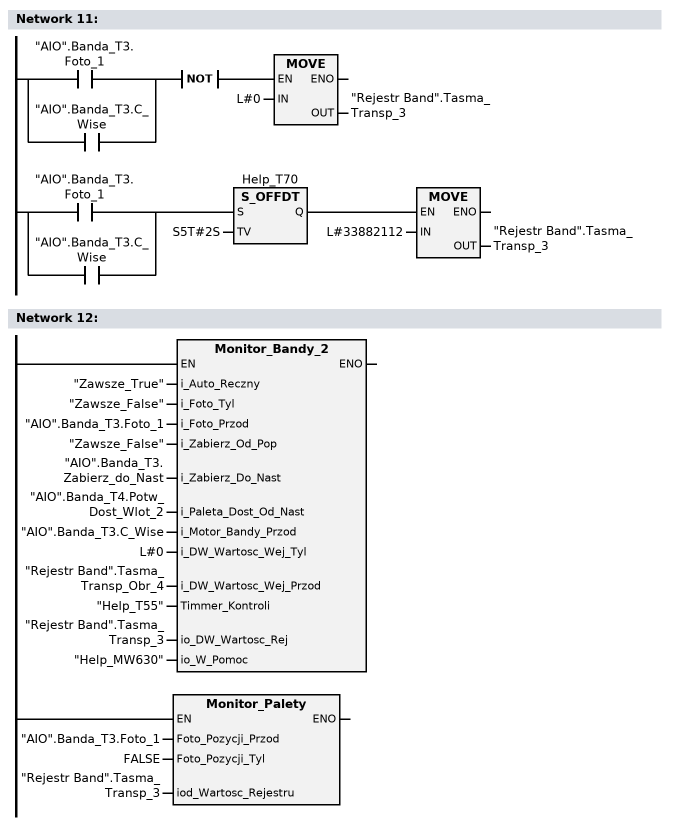
[picture p165: Monitor_Band_Lini networks 11-12]
NETWORK
TITLE =
      O     "AIO".Banda_T3.Foto_1;
      O     "AIO".Banda_T3.C_Wise;
      =     L 1.0;
      A     L 1.0;
      NOT;
      JNB   _003;
      L     L#0;
      T     "Rejestr Band".Tasma_Transp_3;
_003: NOP   0;
      A(;
      A     L 1.0;
      L     S5T#2S;
      SF    "Help_T70";
      NOP   0;
      NOP   0;
      NOP   0;
      A     "Help_T70";
      );
      JNB   _004;
      L     L#33882112;
      T     "Rejestr Band".Tasma_Transp_3;
_004: NOP   0;
NETWORK
TITLE =
//Nastepne monitoringi trzeba dopisac
//How do you do?
//Banda uznawana za wlot 2
//boczna
//Zaladauj wartosc dla wlotu jest to liczba 5 i foliowanie aktywne
//  327 680 -liczba 5
//33 882 112- liczba 5 i foliowanie   (10_0000_0101_0000_0000_0000_0000)
//**********************************************************************
      CALL  "Monitor_Bandy_2" (
           i_Auto_Reczny            := "Zawsze_True",
           i_Foto_Tyl               := "Zawsze_False",
           i_Foto_Przod             := "AIO".Banda_T3.Foto_1,
           i_Zabierz_Od_Pop         := "Zawsze_False",
           i_Zabierz_Do_Nast        := "AIO".Banda_T3.Zabierz_do_Nast,
           i_Paleta_Dost_Od_Nast    := "AIO".Banda_T4.Potw_Dost_Wlot_2,
           i_Motor_Bandy_Przod      := "AIO".Banda_T3.C_Wise,
           i_DW_Wartosc_Wej_Tyl     := L#0,
           i_DW_Wartosc_Wej_Przod   := "Rejestr Band".Tasma_Transp_Obr_4,
           Timmer_Kontroli          := "Help_T55",
           io_DW_Wartosc_Rej        := "Rejestr Band".Tasma_Transp_3,
           io_W_Pomoc               := "Help_MW630");
      CALL  "Monitor_Palety" (
           Foto_Pozycji_Przod       := "AIO".Banda_T3.Foto_1,
           Foto_Pozycji_Tyl         := FALSE,
           iod_Wartosc_Rejestru     := "Rejestr Band".Tasma_Transp_3);
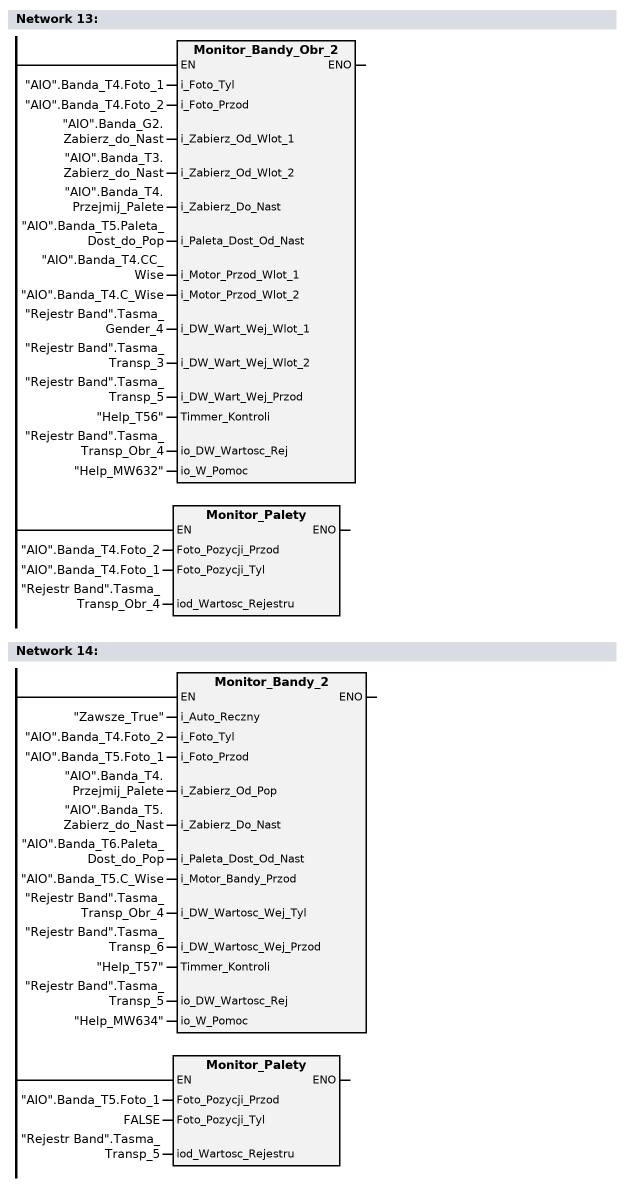
NETWORK
TITLE =
//band a obrotowa T4
//foto_2 to foto blizej foliarki
//motor prawo to motor prosto ("AIO".Banda_T4.CC_Wise)
//motor lewo to motor tyl ("AIO".Banda_T4.C_Wise)
      CALL  "Monitor_Bandy_Obr_2" (
           i_Foto_Tyl               := "AIO".Banda_T4.Foto_1,
           i_Foto_Przod             := "AIO".Banda_T4.Foto_2,
           i_Zabierz_Od_Wlot_1      := "AIO".Banda_G2.Zabierz_do_Nast,
           i_Zabierz_Od_Wlot_2      := "AIO".Banda_T3.Zabierz_do_Nast,
           i_Zabierz_Do_Nast        := "AIO".Banda_T4.Przejmij_Palete,
           i_Paleta_Dost_Od_Nast    := "AIO".Banda_T5.Paleta_Dost_do_Pop,
           i_Motor_Przod_Wlot_1     := "AIO".Banda_T4.CC_Wise,
           i_Motor_Przod_Wlot_2     := "AIO".Banda_T4.C_Wise,
           i_DW_Wart_Wej_Wlot_1     := "Rejestr Band".Tasma_Gender_4,
           i_DW_Wart_Wej_Wlot_2     := "Rejestr Band".Tasma_Transp_3,
           i_DW_Wart_Wej_Przod      := "Rejestr Band".Tasma_Transp_5,
           Timmer_Kontroli          := "Help_T56",
           io_DW_Wartosc_Rej        := "Rejestr Band".Tasma_Transp_Obr_4,
           io_W_Pomoc               := "Help_MW632");
      CALL  "Monitor_Palety" (
           Foto_Pozycji_Przod       := "AIO".Banda_T4.Foto_2,
           Foto_Pozycji_Tyl         := "AIO".Banda_T4.Foto_1,
           iod_Wartosc_Rejestru     := "Rejestr Band".Tasma_Transp_Obr_4);
NETWORK
TITLE =
//Banda T5 foto_2 na obrotnicy to ta blizej foliarki
      CALL  "Monitor_Bandy_2" (
           i_Auto_Reczny            := "Zawsze_True",
           i_Foto_Tyl               := "AIO".Banda_T4.Foto_2,
           i_Foto_Przod             := "AIO".Banda_T5.Foto_1,
           i_Zabierz_Od_Pop         := "AIO".Banda_T4.Przejmij_Palete,
           i_Zabierz_Do_Nast        := "AIO".Banda_T5.Zabierz_do_Nast,
           i_Paleta_Dost_Od_Nast    := "AIO".Banda_T6.Paleta_Dost_do_Pop,
           i_Motor_Bandy_Przod      := "AIO".Banda_T5.C_Wise,
           i_DW_Wartosc_Wej_Tyl     := "Rejestr Band".Tasma_Transp_Obr_4,
           i_DW_Wartosc_Wej_Przod   := "Rejestr Band".Tasma_Transp_6,
           Timmer_Kontroli          := "Help_T57",
           io_DW_Wartosc_Rej        := "Rejestr Band".Tasma_Transp_5,
           io_W_Pomoc               := "Help_MW634");
      CALL  "Monitor_Palety" (
           Foto_Pozycji_Przod       := "AIO".Banda_T5.Foto_1,
           Foto_Pozycji_Tyl         := FALSE,
           iod_Wartosc_Rejestru     := "Rejestr Band".Tasma_Transp_5);
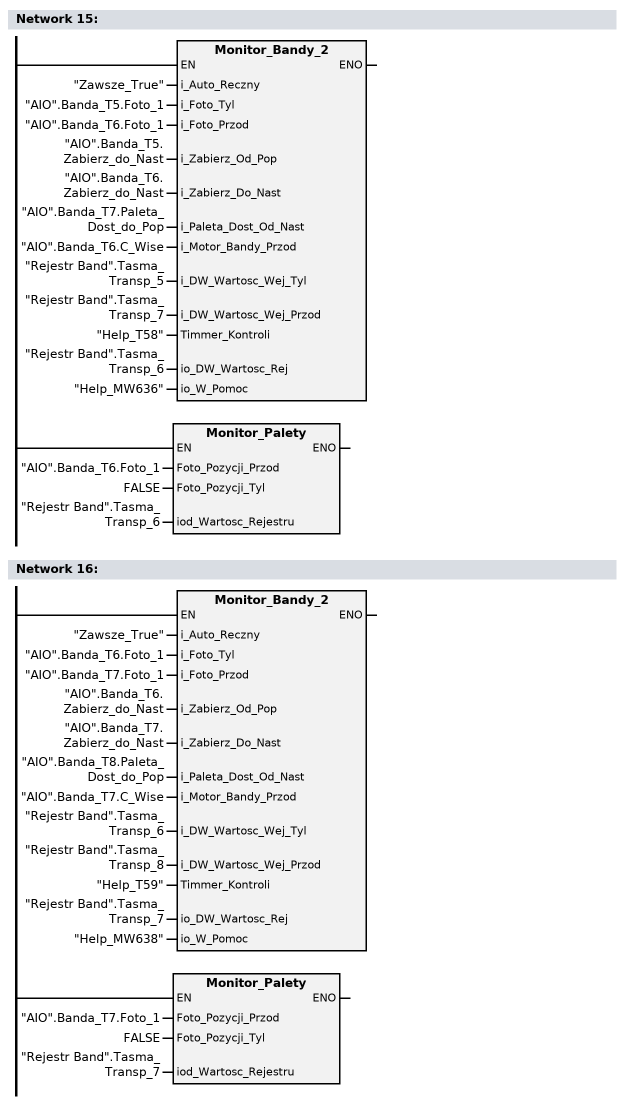
NETWORK
TITLE =
//Banda T6
      CALL  "Monitor_Bandy_2" (
           i_Auto_Reczny            := "Zawsze_True",
           i_Foto_Tyl               := "AIO".Banda_T5.Foto_1,
           i_Foto_Przod             := "AIO".Banda_T6.Foto_1,
           i_Zabierz_Od_Pop         := "AIO".Banda_T5.Zabierz_do_Nast,
           i_Zabierz_Do_Nast        := "AIO".Banda_T6.Zabierz_do_Nast,
           i_Paleta_Dost_Od_Nast    := "AIO".Banda_T7.Paleta_Dost_do_Pop,
           i_Motor_Bandy_Przod      := "AIO".Banda_T6.C_Wise,
           i_DW_Wartosc_Wej_Tyl     := "Rejestr Band".Tasma_Transp_5,
           i_DW_Wartosc_Wej_Przod   := "Rejestr Band".Tasma_Transp_7,
           Timmer_Kontroli          := "Help_T58",
           io_DW_Wartosc_Rej        := "Rejestr Band".Tasma_Transp_6,
           io_W_Pomoc               := "Help_MW636");
      CALL  "Monitor_Palety" (
           Foto_Pozycji_Przod       := "AIO".Banda_T6.Foto_1,
           Foto_Pozycji_Tyl         := FALSE,
           iod_Wartosc_Rejestru     := "Rejestr Band".Tasma_Transp_6);
NETWORK
TITLE =
//Banda T7
//
      CALL  "Monitor_Bandy_2" (
           i_Auto_Reczny            := "Zawsze_True",
           i_Foto_Tyl               := "AIO".Banda_T6.Foto_1,
           i_Foto_Przod             := "AIO".Banda_T7.Foto_1,
           i_Zabierz_Od_Pop         := "AIO".Banda_T6.Zabierz_do_Nast,
           i_Zabierz_Do_Nast        := "AIO".Banda_T7.Zabierz_do_Nast,
           i_Paleta_Dost_Od_Nast    := "AIO".Banda_T8.Paleta_Dost_do_Pop,
           i_Motor_Bandy_Przod      := "AIO".Banda_T7.C_Wise,
           i_DW_Wartosc_Wej_Tyl     := "Rejestr Band".Tasma_Transp_6,
           i_DW_Wartosc_Wej_Przod   := "Rejestr Band".Tasma_Transp_8,
           Timmer_Kontroli          := "Help_T59",
           io_DW_Wartosc_Rej        := "Rejestr Band".Tasma_Transp_7,
           io_W_Pomoc               := "Help_MW638");
      CALL  "Monitor_Palety" (
           Foto_Pozycji_Przod       := "AIO".Banda_T7.Foto_1,
           Foto_Pozycji_Tyl         := FALSE,
           iod_Wartosc_Rejestru     := "Rejestr Band".Tasma_Transp_7);
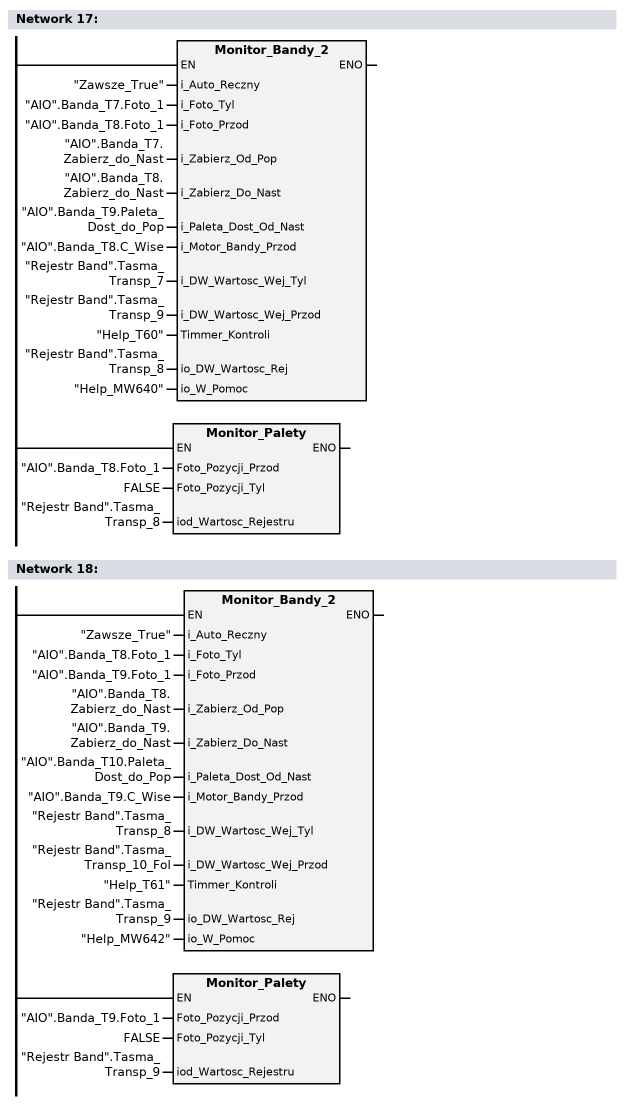
NETWORK
TITLE =
//Banda T8
//
      CALL  "Monitor_Bandy_2" (
           i_Auto_Reczny            := "Zawsze_True",
           i_Foto_Tyl               := "AIO".Banda_T7.Foto_1,
           i_Foto_Przod             := "AIO".Banda_T8.Foto_1,
           i_Zabierz_Od_Pop         := "AIO".Banda_T7.Zabierz_do_Nast,
           i_Zabierz_Do_Nast        := "AIO".Banda_T8.Zabierz_do_Nast,
           i_Paleta_Dost_Od_Nast    := "AIO".Banda_T9.Paleta_Dost_do_Pop,
           i_Motor_Bandy_Przod      := "AIO".Banda_T8.C_Wise,
           i_DW_Wartosc_Wej_Tyl     := "Rejestr Band".Tasma_Transp_7,
           i_DW_Wartosc_Wej_Przod   := "Rejestr Band".Tasma_Transp_9,
           Timmer_Kontroli          := "Help_T60",
           io_DW_Wartosc_Rej        := "Rejestr Band".Tasma_Transp_8,
           io_W_Pomoc               := "Help_MW640");
      CALL  "Monitor_Palety" (
           Foto_Pozycji_Przod       := "AIO".Banda_T8.Foto_1,
           Foto_Pozycji_Tyl         := FALSE,
           iod_Wartosc_Rejestru     := "Rejestr Band".Tasma_Transp_8);
NETWORK
TITLE =
//Banda T9
//
      CALL  "Monitor_Bandy_2" (
           i_Auto_Reczny            := "Zawsze_True",
           i_Foto_Tyl               := "AIO".Banda_T8.Foto_1,
           i_Foto_Przod             := "AIO".Banda_T9.Foto_1,
           i_Zabierz_Od_Pop         := "AIO".Banda_T8.Zabierz_do_Nast,
           i_Zabierz_Do_Nast        := "AIO".Banda_T9.Zabierz_do_Nast,
           i_Paleta_Dost_Od_Nast    := "AIO".Banda_T10.Paleta_Dost_do_Pop,
           i_Motor_Bandy_Przod      := "AIO".Banda_T9.C_Wise,
           i_DW_Wartosc_Wej_Tyl     := "Rejestr Band".Tasma_Transp_8,
           i_DW_Wartosc_Wej_Przod   := "Rejestr Band".Tasma_Transp_10_Fol,
           Timmer_Kontroli          := "Help_T61",
           io_DW_Wartosc_Rej        := "Rejestr Band".Tasma_Transp_9,
           io_W_Pomoc               := "Help_MW642");
      CALL  "Monitor_Palety" (
           Foto_Pozycji_Przod       := "AIO".Banda_T9.Foto_1,
           Foto_Pozycji_Tyl         := FALSE,
           iod_Wartosc_Rejestru     := "Rejestr Band".Tasma_Transp_9);
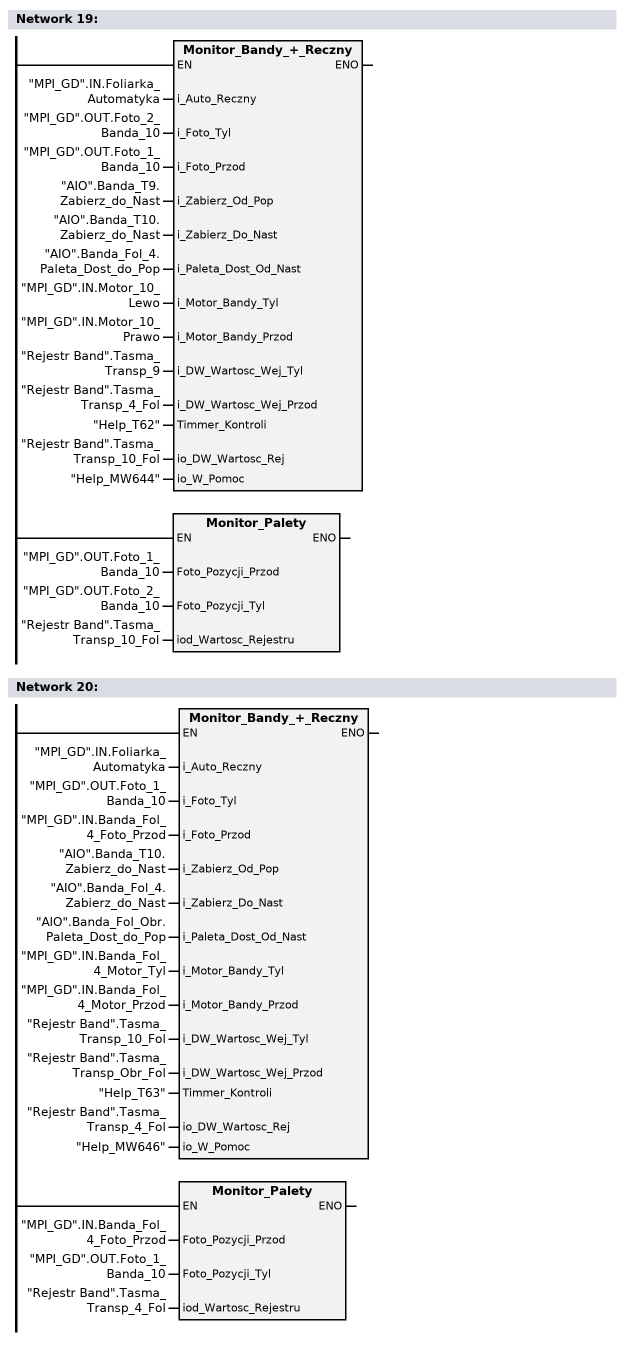
NETWORK
TITLE =
//Banda T10 - Banda 2 foliarka (ta banda jest wspolna dla lini transportowej i 
//foliarki)
//
//
//
      CALL  "Monitor_Bandy_+_Reczny" (
           i_Auto_Reczny            := "MPI_GD".IN.Foliarka_Automatyka,
           i_Foto_Tyl               := "MPI_GD".OUT.Foto_2_Banda_10,
           i_Foto_Przod             := "MPI_GD".OUT.Foto_1_Banda_10,
           i_Zabierz_Od_Pop         := "AIO".Banda_T9.Zabierz_do_Nast,
           i_Zabierz_Do_Nast        := "AIO".Banda_T10.Zabierz_do_Nast,
           i_Paleta_Dost_Od_Nast    := "AIO".Banda_Fol_4.Paleta_Dost_do_Pop,
           i_Motor_Bandy_Tyl        := "MPI_GD".IN.Motor_10_Lewo,
           i_Motor_Bandy_Przod      := "MPI_GD".IN.Motor_10_Prawo,
           i_DW_Wartosc_Wej_Tyl     := "Rejestr Band".Tasma_Transp_9,
           i_DW_Wartosc_Wej_Przod   := "Rejestr Band".Tasma_Transp_4_Fol,
           Timmer_Kontroli          := "Help_T62",
           io_DW_Wartosc_Rej        := "Rejestr Band".Tasma_Transp_10_Fol,
           io_W_Pomoc               := "Help_MW644");
      CALL  "Monitor_Palety" (
           Foto_Pozycji_Przod       := "MPI_GD".OUT.Foto_1_Banda_10,
           Foto_Pozycji_Tyl         := "MPI_GD".OUT.Foto_2_Banda_10,
           iod_Wartosc_Rejestru     := "Rejestr Band".Tasma_Transp_10_Fol);
NETWORK
TITLE =
//Banda Virtulana foliarki 4
//
      CALL  "Monitor_Bandy_+_Reczny" (
           i_Auto_Reczny            := "MPI_GD".IN.Foliarka_Automatyka,
           i_Foto_Tyl               := "MPI_GD".OUT.Foto_1_Banda_10,
           i_Foto_Przod             := "MPI_GD".IN.Banda_Fol_4_Foto_Przod,
           i_Zabierz_Od_Pop         := "AIO".Banda_T10.Zabierz_do_Nast,
           i_Zabierz_Do_Nast        := "AIO".Banda_Fol_4.Zabierz_do_Nast,
           i_Paleta_Dost_Od_Nast    := "AIO".Banda_Fol_Obr.Paleta_Dost_do_Pop,
           i_Motor_Bandy_Tyl        := "MPI_GD".IN.Banda_Fol_4_Motor_Tyl,
           i_Motor_Bandy_Przod      := "MPI_GD".IN.Banda_Fol_4_Motor_Przod,
           i_DW_Wartosc_Wej_Tyl     := "Rejestr Band".Tasma_Transp_10_Fol,
           i_DW_Wartosc_Wej_Przod   := "Rejestr Band".Tasma_Transp_Obr_Fol,
           Timmer_Kontroli          := "Help_T63",
           io_DW_Wartosc_Rej        := "Rejestr Band".Tasma_Transp_4_Fol,
           io_W_Pomoc               := "Help_MW646");
      CALL  "Monitor_Palety" (
           Foto_Pozycji_Przod       := "MPI_GD".IN.Banda_Fol_4_Foto_Przod,
           Foto_Pozycji_Tyl         := "MPI_GD".OUT.Foto_1_Banda_10,
           iod_Wartosc_Rejestru     := "Rejestr Band".Tasma_Transp_4_Fol);
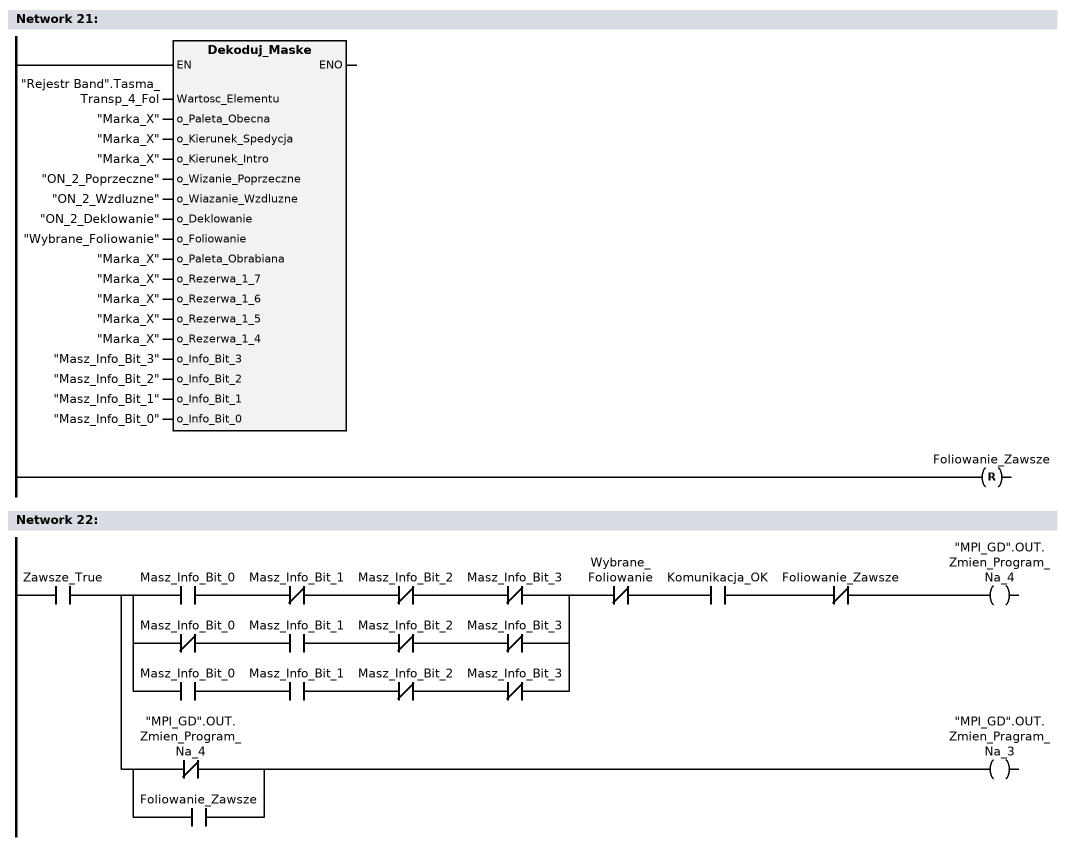
NETWORK
TITLE =
//Dekodowanie maski. Aby umozliwic bindowanie
//-Obsluga wiazan jest w FC120
//-Obsluga Dekla jest w FB3
//
      CALL  "Dekoduj_Maske" (
           Wartosc_Elementu         := "Rejestr Band".Tasma_Transp_4_Fol,
           o_Paleta_Obecna          := "Marka_X",
           o_Kierunek_Spedycja      := "Marka_X",
           o_Kierunek_Intro         := "Marka_X",
           o_Wizanie_Poprzeczne     := "ON_2_Poprzeczne",
           o_Wiazanie_Wzdluzne      := "ON_2_Wzdluzne",
           o_Deklowanie             := "ON_2_Deklowanie",
           o_Foliowanie             := "Wybrane_Foliowanie",
           o_Paleta_Obrabiana       := "Marka_X",
           o_Rezerwa_1_7            := "Marka_X",
           o_Rezerwa_1_6            := "Marka_X",
           o_Rezerwa_1_5            := "Marka_X",
           o_Rezerwa_1_4            := "Marka_X",
           o_Info_Bit_3             := "Masz_Info_Bit_3",
           o_Info_Bit_2             := "Masz_Info_Bit_2",
           o_Info_Bit_1             := "Masz_Info_Bit_1",
           o_Info_Bit_0             := "Masz_Info_Bit_0");
//Zmien program na program 4
      SET;
      R     "Foliowanie_Zawsze";
NETWORK
TITLE =
//Wybor programu foliujacego. Przewaga foliowania nad brakiem foliowania. 
//Brak foliowania wystapi jedynie gdy bedzie brak foliowania na kolbusie 1,2 oraz 
//bufforach.Po za tym paleta nie moze stracic miejsca pochodzenia
//
      A     "Zawsze_True";
      =     L 1.0;
      A     L 1.0;
      A(;
      A     "Masz_Info_Bit_0";
      AN    "Masz_Info_Bit_1";
      AN    "Masz_Info_Bit_2";
      AN    "Masz_Info_Bit_3";
      O;
      AN    "Masz_Info_Bit_0";
      A     "Masz_Info_Bit_1";
      AN    "Masz_Info_Bit_2";
      AN    "Masz_Info_Bit_3";
      O;
      A     "Masz_Info_Bit_0";
      A     "Masz_Info_Bit_1";
      AN    "Masz_Info_Bit_2";
      AN    "Masz_Info_Bit_3";
      );
      AN    "Wybrane_Foliowanie";
      A     "Komunikacja_OK";
      AN    "Foliowanie_Zawsze";
      =     "MPI_GD".OUT.Zmien_Program_Na_4;
      A     L 1.0;
      A(;
      ON    "MPI_GD".OUT.Zmien_Program_Na_4;
      O     "Foliowanie_Zawsze";
      );
      =     "MPI_GD".OUT.Zmien_Pragram_Na_3;
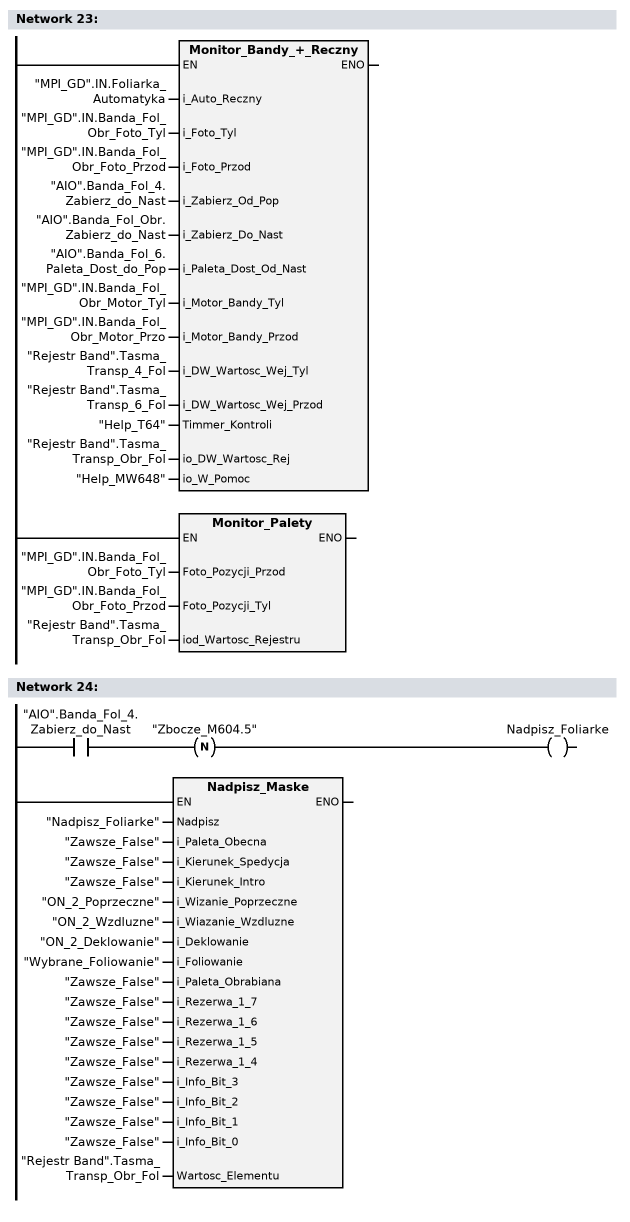
NETWORK
TITLE =
//Banda Virtulana foliarki obr
//
      CALL  "Monitor_Bandy_+_Reczny" (
           i_Auto_Reczny            := "MPI_GD".IN.Foliarka_Automatyka,
           i_Foto_Tyl               := "MPI_GD".IN.Banda_Fol_Obr_Foto_Tyl,
           i_Foto_Przod             := "MPI_GD".IN.Banda_Fol_Obr_Foto_Przod,
           i_Zabierz_Od_Pop         := "AIO".Banda_Fol_4.Zabierz_do_Nast,
           i_Zabierz_Do_Nast        := "AIO".Banda_Fol_Obr.Zabierz_do_Nast,
           i_Paleta_Dost_Od_Nast    := "AIO".Banda_Fol_6.Paleta_Dost_do_Pop,
           i_Motor_Bandy_Tyl        := "MPI_GD".IN.Banda_Fol_Obr_Motor_Tyl,
           i_Motor_Bandy_Przod      := "MPI_GD".IN.Banda_Fol_Obr_Motor_Przo,
           i_DW_Wartosc_Wej_Tyl     := "Rejestr Band".Tasma_Transp_4_Fol,
           i_DW_Wartosc_Wej_Przod   := "Rejestr Band".Tasma_Transp_6_Fol,
           Timmer_Kontroli          := "Help_T64",
           io_DW_Wartosc_Rej        := "Rejestr Band".Tasma_Transp_Obr_Fol,
           io_W_Pomoc               := "Help_MW648");
      CALL  "Monitor_Palety" (
           Foto_Pozycji_Przod       := "MPI_GD".IN.Banda_Fol_Obr_Foto_Tyl,
           Foto_Pozycji_Tyl         := "MPI_GD".IN.Banda_Fol_Obr_Foto_Przod,
           iod_Wartosc_Rejestru     := "Rejestr Band".Tasma_Transp_Obr_Fol);
NETWORK
TITLE =
//Nadpisz Maske
      A     "AIO".Banda_Fol_4.Zabierz_do_Nast;
      FN    "Zbocze_M604.5";
      =     "Nadpisz_Foliarke";
      CALL  "Nadpisz_Maske" (
           Nadpisz                  := "Nadpisz_Foliarke",
           i_Paleta_Obecna          := "Zawsze_False",
           i_Kierunek_Spedycja      := "Zawsze_False",
           i_Kierunek_Intro         := "Zawsze_False",
           i_Wizanie_Poprzeczne     := "ON_2_Poprzeczne",
           i_Wiazanie_Wzdluzne      := "ON_2_Wzdluzne",
           i_Deklowanie             := "ON_2_Deklowanie",
           i_Foliowanie             := "Wybrane_Foliowanie",
           i_Paleta_Obrabiana       := "Zawsze_False",
           i_Rezerwa_1_7            := "Zawsze_False",
           i_Rezerwa_1_6            := "Zawsze_False",
           i_Rezerwa_1_5            := "Zawsze_False",
           i_Rezerwa_1_4            := "Zawsze_False",
           i_Info_Bit_3             := "Zawsze_False",
           i_Info_Bit_2             := "Zawsze_False",
           i_Info_Bit_1             := "Zawsze_False",
           i_Info_Bit_0             := "Zawsze_False",
           Wartosc_Elementu         := "Rejestr Band".Tasma_Transp_Obr_Fol);
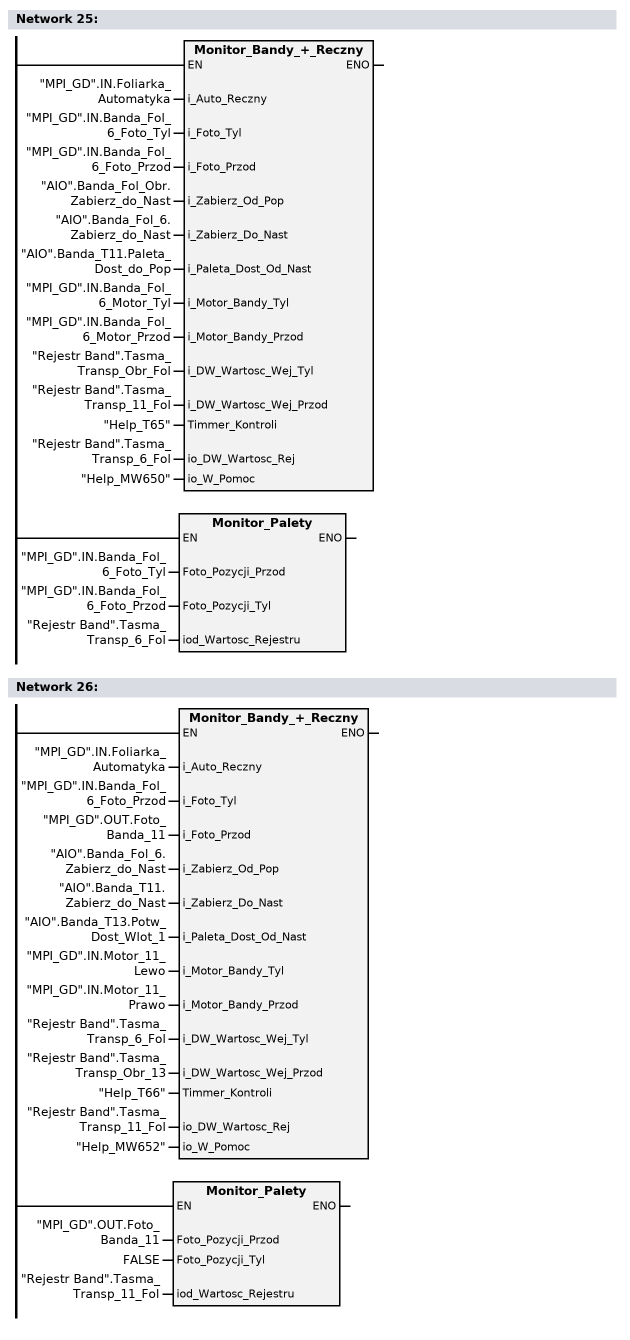
NETWORK
TITLE =
//Banda Virtulana foliarki 6
//
      CALL  "Monitor_Bandy_+_Reczny" (
           i_Auto_Reczny            := "MPI_GD".IN.Foliarka_Automatyka,
           i_Foto_Tyl               := "MPI_GD".IN.Banda_Fol_6_Foto_Tyl,
           i_Foto_Przod             := "MPI_GD".IN.Banda_Fol_6_Foto_Przod,
           i_Zabierz_Od_Pop         := "AIO".Banda_Fol_Obr.Zabierz_do_Nast,
           i_Zabierz_Do_Nast        := "AIO".Banda_Fol_6.Zabierz_do_Nast,
           i_Paleta_Dost_Od_Nast    := "AIO".Banda_T11.Paleta_Dost_do_Pop,
           i_Motor_Bandy_Tyl        := "MPI_GD".IN.Banda_Fol_6_Motor_Tyl,
           i_Motor_Bandy_Przod      := "MPI_GD".IN.Banda_Fol_6_Motor_Przod,
           i_DW_Wartosc_Wej_Tyl     := "Rejestr Band".Tasma_Transp_Obr_Fol,
           i_DW_Wartosc_Wej_Przod   := "Rejestr Band".Tasma_Transp_11_Fol,
           Timmer_Kontroli          := "Help_T65",
           io_DW_Wartosc_Rej        := "Rejestr Band".Tasma_Transp_6_Fol,
           io_W_Pomoc               := "Help_MW650");
      CALL  "Monitor_Palety" (
           Foto_Pozycji_Przod       := "MPI_GD".IN.Banda_Fol_6_Foto_Tyl,
           Foto_Pozycji_Tyl         := "MPI_GD".IN.Banda_Fol_6_Foto_Przod,
           iod_Wartosc_Rejestru     := "Rejestr Band".Tasma_Transp_6_Fol);
NETWORK
TITLE =
//Banda foliarki 11 wspolna z linia
//
      CALL  "Monitor_Bandy_+_Reczny" (
           i_Auto_Reczny            := "MPI_GD".IN.Foliarka_Automatyka,
           i_Foto_Tyl               := "MPI_GD".IN.Banda_Fol_6_Foto_Przod,
           i_Foto_Przod             := "MPI_GD".OUT.Foto_Banda_11,
           i_Zabierz_Od_Pop         := "AIO".Banda_Fol_6.Zabierz_do_Nast,
           i_Zabierz_Do_Nast        := "AIO".Banda_T11.Zabierz_do_Nast,
           i_Paleta_Dost_Od_Nast    := "AIO".Banda_T13.Potw_Dost_Wlot_1,
           i_Motor_Bandy_Tyl        := "MPI_GD".IN.Motor_11_Lewo,
           i_Motor_Bandy_Przod      := "MPI_GD".IN.Motor_11_Prawo,
           i_DW_Wartosc_Wej_Tyl     := "Rejestr Band".Tasma_Transp_6_Fol,
           i_DW_Wartosc_Wej_Przod   := "Rejestr Band".Tasma_Transp_Obr_13,
           Timmer_Kontroli          := "Help_T66",
           io_DW_Wartosc_Rej        := "Rejestr Band".Tasma_Transp_11_Fol,
           io_W_Pomoc               := "Help_MW652");
      CALL  "Monitor_Palety" (
           Foto_Pozycji_Przod       := "MPI_GD".OUT.Foto_Banda_11,
           Foto_Pozycji_Tyl         := FALSE,
           iod_Wartosc_Rejestru     := "Rejestr Band".Tasma_Transp_11_Fol);
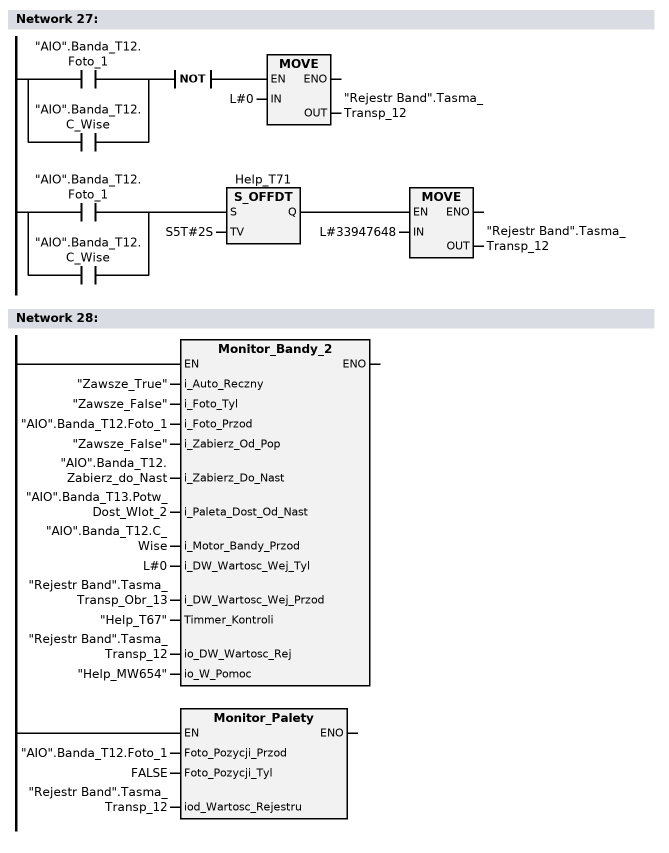
NETWORK
TITLE =
      O     "AIO".Banda_T12.Foto_1;
      O     "AIO".Banda_T12.C_Wise;
      =     L 1.0;
      A     L 1.0;
      NOT;
      JNB   _005;
      L     L#0;
      T     "Rejestr Band".Tasma_Transp_12;
_005: NOP   0;
      A(;
      A     L 1.0;
      L     S5T#2S;
      SF    "Help_T71";
      NOP   0;
      NOP   0;
      NOP   0;
      A     "Help_T71";
      );
      JNB   _006;
      L     L#33947648;
      T     "Rejestr Band".Tasma_Transp_12;
_006: NOP   0;
NETWORK
TITLE =
//Nastepne monitoringi trzeba dopisac
//Banda uznawana za wlot 3
//boczna
//Zaladauj wartosc dla wlotu jest to liczba 5 i foliowanie aktywne
//33 947 648- liczba 6 i foliowanie   (10_0000_0110_0000_0000_0000_0000)
//**********************************************************************
      CALL  "Monitor_Bandy_2" (
           i_Auto_Reczny            := "Zawsze_True",
           i_Foto_Tyl               := "Zawsze_False",
           i_Foto_Przod             := "AIO".Banda_T12.Foto_1,
           i_Zabierz_Od_Pop         := "Zawsze_False",
           i_Zabierz_Do_Nast        := "AIO".Banda_T12.Zabierz_do_Nast,
           i_Paleta_Dost_Od_Nast    := "AIO".Banda_T13.Potw_Dost_Wlot_2,
           i_Motor_Bandy_Przod      := "AIO".Banda_T12.C_Wise,
           i_DW_Wartosc_Wej_Tyl     := L#0,
           i_DW_Wartosc_Wej_Przod   := "Rejestr Band".Tasma_Transp_Obr_13,
           Timmer_Kontroli          := "Help_T67",
           io_DW_Wartosc_Rej        := "Rejestr Band".Tasma_Transp_12,
           io_W_Pomoc               := "Help_MW654");
      CALL  "Monitor_Palety" (
           Foto_Pozycji_Przod       := "AIO".Banda_T12.Foto_1,
           Foto_Pozycji_Tyl         := FALSE,
           iod_Wartosc_Rejestru     := "Rejestr Band".Tasma_Transp_12);
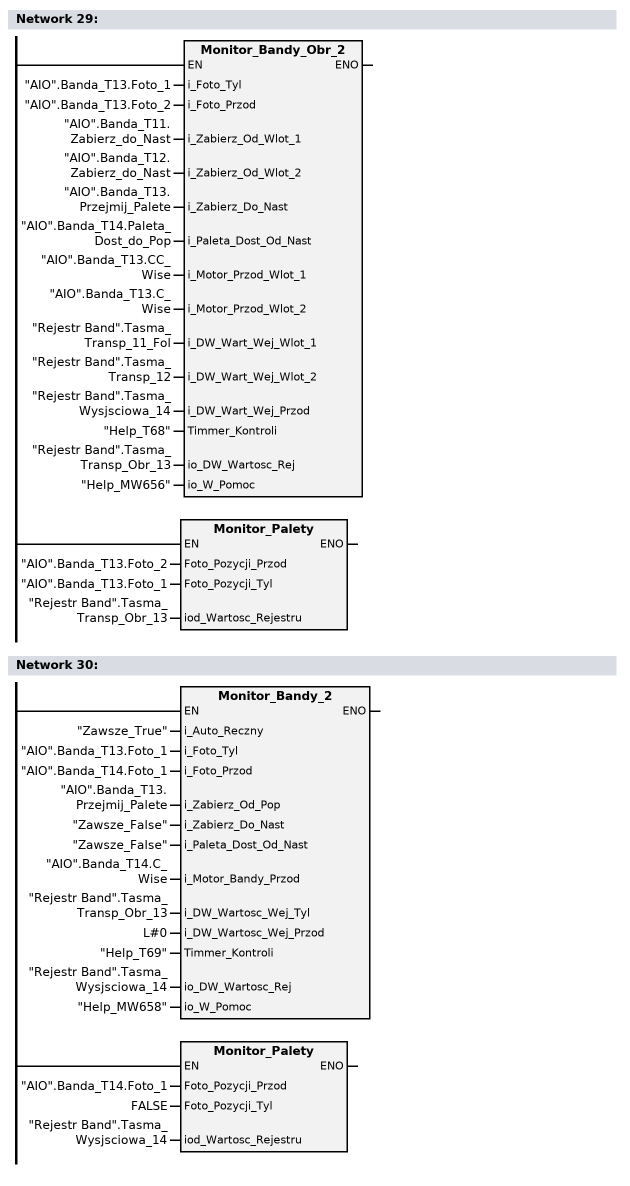
NETWORK
TITLE =
//Banda Obrotowa
//foto_2 to przod od foliarki i motor prawo
      CALL  "Monitor_Bandy_Obr_2" (
           i_Foto_Tyl               := "AIO".Banda_T13.Foto_1,
           i_Foto_Przod             := "AIO".Banda_T13.Foto_2,
           i_Zabierz_Od_Wlot_1      := "AIO".Banda_T11.Zabierz_do_Nast,
           i_Zabierz_Od_Wlot_2      := "AIO".Banda_T12.Zabierz_do_Nast,
           i_Zabierz_Do_Nast        := "AIO".Banda_T13.Przejmij_Palete,
           i_Paleta_Dost_Od_Nast    := "AIO".Banda_T14.Paleta_Dost_do_Pop,
           i_Motor_Przod_Wlot_1     := "AIO".Banda_T13.CC_Wise,
           i_Motor_Przod_Wlot_2     := "AIO".Banda_T13.C_Wise,
           i_DW_Wart_Wej_Wlot_1     := "Rejestr Band".Tasma_Transp_11_Fol,
           i_DW_Wart_Wej_Wlot_2     := "Rejestr Band".Tasma_Transp_12,
           i_DW_Wart_Wej_Przod      := "Rejestr Band".Tasma_Wysjsciowa_14,
           Timmer_Kontroli          := "Help_T68",
           io_DW_Wartosc_Rej        := "Rejestr Band".Tasma_Transp_Obr_13,
           io_W_Pomoc               := "Help_MW656");
      CALL  "Monitor_Palety" (
           Foto_Pozycji_Przod       := "AIO".Banda_T13.Foto_2,
           Foto_Pozycji_Tyl         := "AIO".Banda_T13.Foto_1,
           iod_Wartosc_Rejestru     := "Rejestr Band".Tasma_Transp_Obr_13);
NETWORK
TITLE =
//Banda Wyjsciowa ostatnia. Danke schon.
      CALL  "Monitor_Bandy_2" (
           i_Auto_Reczny            := "Zawsze_True",
           i_Foto_Tyl               := "AIO".Banda_T13.Foto_1,
           i_Foto_Przod             := "AIO".Banda_T14.Foto_1,
           i_Zabierz_Od_Pop         := "AIO".Banda_T13.Przejmij_Palete,
           i_Zabierz_Do_Nast        := "Zawsze_False",
           i_Paleta_Dost_Od_Nast    := "Zawsze_False",
           i_Motor_Bandy_Przod      := "AIO".Banda_T14.C_Wise,
           i_DW_Wartosc_Wej_Tyl     := "Rejestr Band".Tasma_Transp_Obr_13,
           i_DW_Wartosc_Wej_Przod   := L#0,
           Timmer_Kontroli          := "Help_T69",
           io_DW_Wartosc_Rej        := "Rejestr Band".Tasma_Wysjsciowa_14,
           io_W_Pomoc               := "Help_MW658");
      CALL  "Monitor_Palety" (
           Foto_Pozycji_Przod       := "AIO".Banda_T14.Foto_1,
           Foto_Pozycji_Tyl         := FALSE,
           iod_Wartosc_Rejestru     := "Rejestr Band".Tasma_Wysjsciowa_14);
END_FUNCTION

FUNCTION "Monitor_Bandy" : VOID	// FC 313
//Funkcja na monitoruje przejezdzajacy miedzy bandami produkt
VERSION : 0.1
VAR_INPUT
  i_Foto_Koniec : BOOL ;
  i_Motor_Bandy : BOOL ;
  i_Zabierz_Od_Pop : BOOL ;	//Sygnal zabierz od bandy poprzedniej
  i_Zabierz_Do_Nast : BOOL ;	//Sygnal zabierz do nastepnej
  i_DW_Wartosc_Wej : DINT ;	//Wartosc wejsciowa z poprzedniej bandy
  i_Paleta_Dost_Od_Nast : BOOL ;
END_VAR
VAR_IN_OUT
  io_DW_Wartosc_Rej : DINT ;	//Wartosc bierzaca rejestru
  io_W_Pomoc : WORD ;	//Slowo pomocnicze
END_VAR
VAR_TEMP
  Rel_Z_Pop_Aktywna : BOOL ;	//Relacja z banda poprzednia jest aktywna
  Rel_Z_Nast_Aktywna : BOOL ;	//Relacja z banda nastepna jest aktywan
  Pom_LB1 : BYTE ;
  Pom_LW2 : WORD ;
  Pom_LD4 : BOOL ;
END_VAR
BEGIN
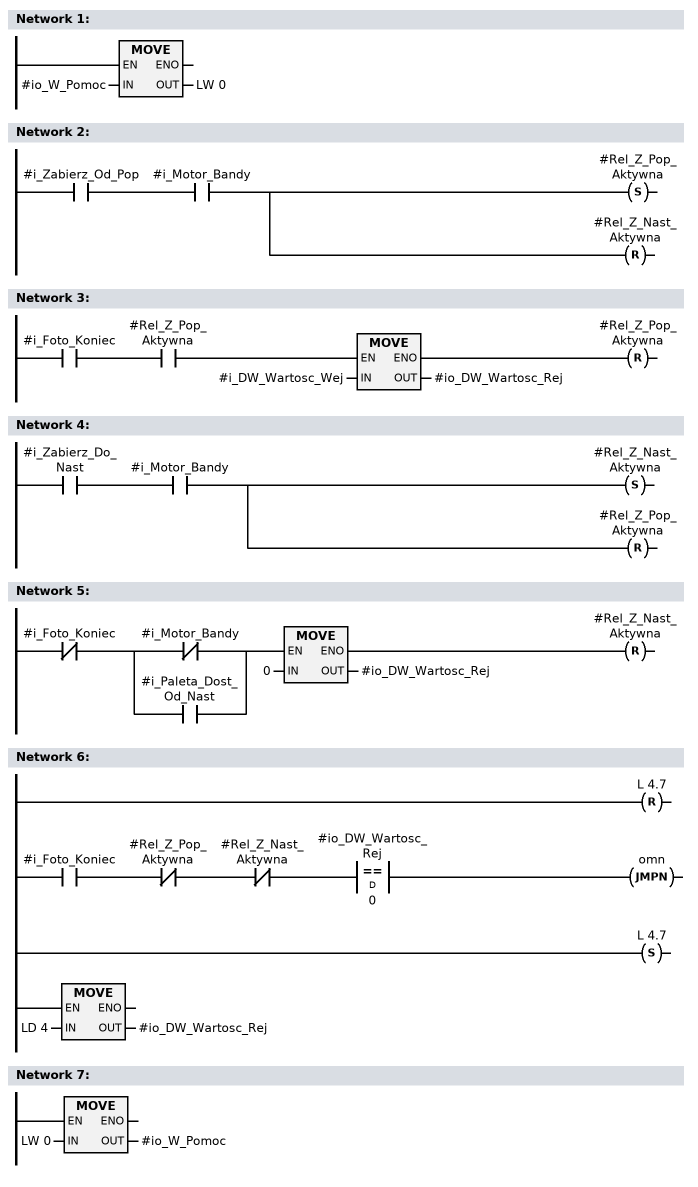
NETWORK
TITLE =
//Ten network celowo jest wolny
      L     #io_W_Pomoc;
      T     LW 0;
      NOP   0;
NETWORK
TITLE =
//Pobranie wartosci
      A     #i_Zabierz_Od_Pop;
      A     #i_Motor_Bandy;
      S     #Rel_Z_Pop_Aktywna;
      R     #Rel_Z_Nast_Aktywna;
NETWORK
TITLE =
//Dojazd do fotokomorki i przepisanie wartosci
      A     #i_Foto_Koniec;
      A     #Rel_Z_Pop_Aktywna;
      JNB   _001;
      L     #i_DW_Wartosc_Wej;
      T     #io_DW_Wartosc_Rej;
      SET;
      SAVE;
      CLR;
_001: A     BR;
      R     #Rel_Z_Pop_Aktywna;
NETWORK
TITLE =
//Relacja z nastepna banda
      A     #i_Zabierz_Do_Nast;
      A     #i_Motor_Bandy;
      S     #Rel_Z_Nast_Aktywna;
      R     #Rel_Z_Pop_Aktywna;
NETWORK
TITLE =
//Opuszczeni palety z bandy relacja przod
      AN    #i_Foto_Koniec;
      A(;
      ON    #i_Motor_Bandy;
      O     #i_Paleta_Dost_Od_Nast;
      );
      JNB   _002;
      L     0;
      T     #io_DW_Wartosc_Rej;
      SET;
      SAVE;
      CLR;
_002: A     BR;
      R     #Rel_Z_Nast_Aktywna;
NETWORK
TITLE =
//Nalozenie maski gdy jest paleta a wartosc rejsetru wskazuje na 0
//kasowanie bitu pomocniczego
      SET;
      R     L 4.7;
// Aby znalezc palete widmo
      A     #i_Foto_Koniec;
      AN    #Rel_Z_Pop_Aktywna;
      AN    #Rel_Z_Nast_Aktywna;
      A(;
      L     #io_DW_Wartosc_Rej;
      L     0;
      ==D;
      );
      JCN   omn;
      SET;
      S     L 4.7;	//najstarszy bit (info o palecie)
      L     LD 4;
      T     #io_DW_Wartosc_Rej;
omn:  NOP   0;
NETWORK
TITLE =
//Przypisanie wartosci z pamieci podrecznej
//
      L     LW 0;
      T     #io_W_Pomoc;
      NOP   0;
END_FUNCTION

FUNCTION "Monitor_Bandy_Obr" : VOID	// FC 314
//Funkcja na monitoruje przejezdzajacy miedzy bandami produkt
VERSION : 0.1
VAR_INPUT
  i_Foto_Koniec_Wlot_1 : BOOL ;
  i_Foto_Koniec_Wlot_2 : BOOL ;
  i_Foto_Koniec_Wylot : BOOL ;
  i_Motor_Bandy : BOOL ;
  i_Zabierz_Od_Wlot_1 : BOOL ;	//Sygnal zabierz od bandy poprzedniej
  i_Zabierz_Od_Wlot_2 : BOOL ;	//Sygnal zabierz od bandy poprzedniej
  i_Zabierz_Do_Nast : BOOL ;	//Sygnal zabierz do nastepnej
  i_DW_Wart_Wej_Wlot_1 : DINT ;	//Wartosc wejsciowa z wlotu 1
  i_DW_Wart_Wej_Wlot_2 : DINT ;	//Wartosc wejsciowa z wlotu 2
  i_Paleta_Dost_Od_Nast : BOOL ;
END_VAR
VAR_IN_OUT
  io_DW_Wartosc_Rej : DINT ;	//Wartosc bierzaca rejestru
  io_W_Pomoc : WORD ;	//Slowo pomocnicze
END_VAR
VAR_TEMP
  Rel_Aktyw_z_Wlot_1 : BOOL ;	//Relacja z banda poprzednia jest aktywna
  Rel_Aktyw_z_Wlot_2 : BOOL ;	//Relacja z banda poprzednia jest aktywna
  Rel_Z_Nast_Aktywna : BOOL ;	//Relacja z banda nastepna jest aktywan
  Pom_LB1 : BYTE ;
  Pom_LW2 : WORD ;
  Pom_LD4 : DINT ;
END_VAR
BEGIN
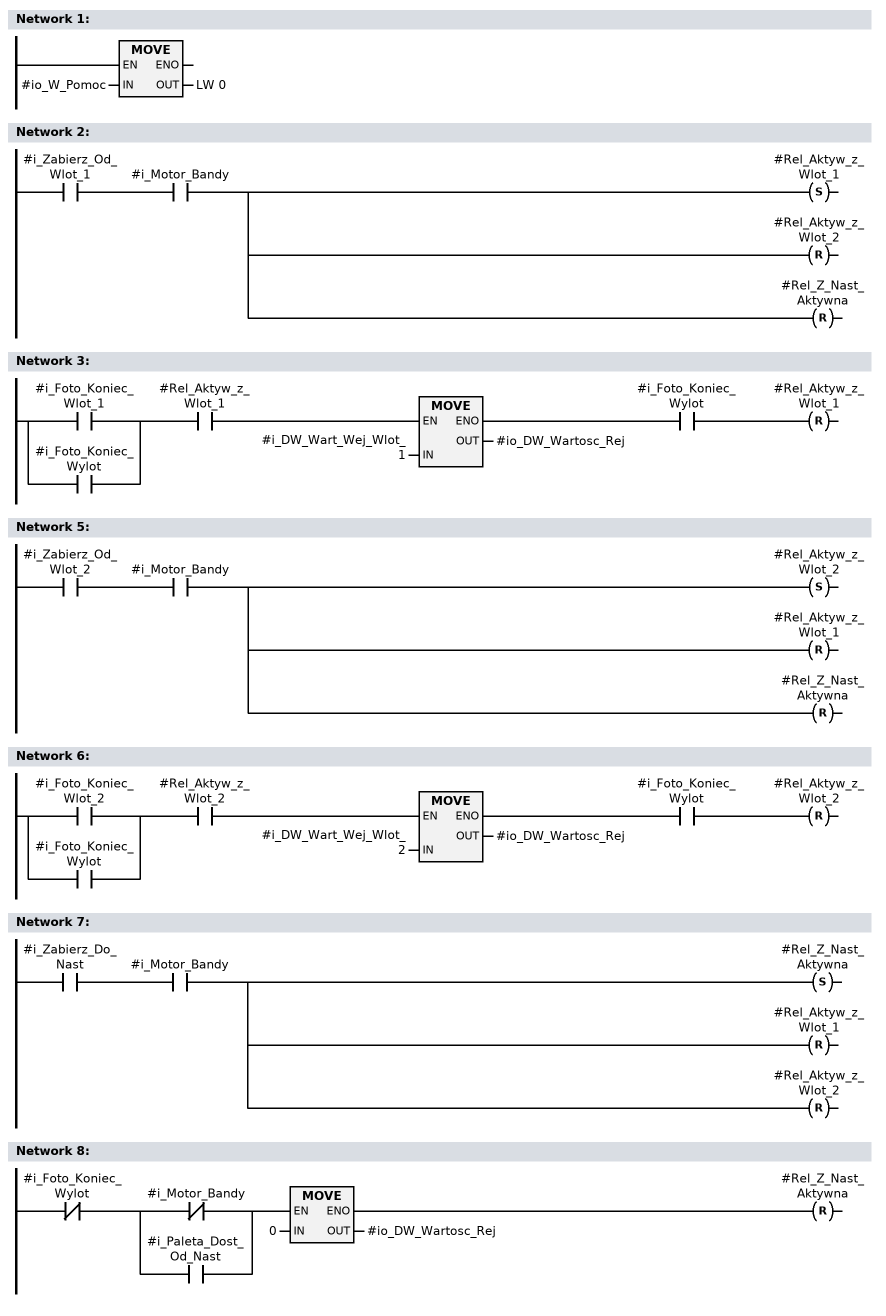
NETWORK
TITLE =
//Ten network celowo jest wolny
      L     #io_W_Pomoc;
      T     LW 0;
      NOP   0;
NETWORK
TITLE =
//Sprawdzenie Relacji z wolotem nr 1
      A     #i_Zabierz_Od_Wlot_1;
      A     #i_Motor_Bandy;
      S     #Rel_Aktyw_z_Wlot_1;
      R     #Rel_Aktyw_z_Wlot_2;
      R     #Rel_Z_Nast_Aktywna;
NETWORK
TITLE =
//Dojazd do fotokomorki i przepisanie wartosci
      A(;
      A(;
      O     #i_Foto_Koniec_Wlot_1;
      O     #i_Foto_Koniec_Wylot;
      );
      A     #Rel_Aktyw_z_Wlot_1;
      JNB   _001;
      L     #i_DW_Wart_Wej_Wlot_1;
      T     #io_DW_Wartosc_Rej;
      SET;
      SAVE;
      CLR;
_001: A     BR;
      );
      A     #i_Foto_Koniec_Wylot;
      R     #Rel_Aktyw_z_Wlot_1;
NETWORK
TITLE =
//Relacja z wlotem nr 2
NETWORK
TITLE =
//Sprawdzenie Relacji z wolotem nr 2
      A     #i_Zabierz_Od_Wlot_2;
      A     #i_Motor_Bandy;
      S     #Rel_Aktyw_z_Wlot_2;
      R     #Rel_Aktyw_z_Wlot_1;
      R     #Rel_Z_Nast_Aktywna;
NETWORK
TITLE =
//Dojazd do fotokomorki i przepisanie wartosci
      A(;
      A(;
      O     #i_Foto_Koniec_Wlot_2;
      O     #i_Foto_Koniec_Wylot;
      );
      A     #Rel_Aktyw_z_Wlot_2;
      JNB   _002;
      L     #i_DW_Wart_Wej_Wlot_2;
      T     #io_DW_Wartosc_Rej;
      SET;
      SAVE;
      CLR;
_002: A     BR;
      );
      A     #i_Foto_Koniec_Wylot;
      R     #Rel_Aktyw_z_Wlot_2;
NETWORK
TITLE =
//Relacja z nastepna banda
      A     #i_Zabierz_Do_Nast;
      A     #i_Motor_Bandy;
      S     #Rel_Z_Nast_Aktywna;
      R     #Rel_Aktyw_z_Wlot_1;
      R     #Rel_Aktyw_z_Wlot_2;
NETWORK
TITLE =
//Opuszczeni palety z bandy relacja przod
      AN    #i_Foto_Koniec_Wylot;
      A(;
      ON    #i_Motor_Bandy;
      O     #i_Paleta_Dost_Od_Nast;
      );
      JNB   _003;
      L     0;
      T     #io_DW_Wartosc_Rej;
      SET;
      SAVE;
      CLR;
_003: A     BR;
      R     #Rel_Z_Nast_Aktywna;
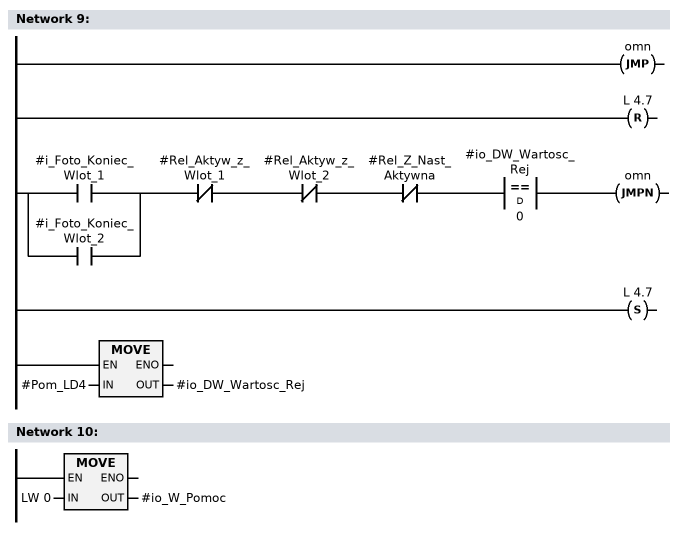
NETWORK
TITLE =
//Nalozenie maski gdy jest paleta a wartosc rejsetru wskazuje na 0
//kasowanie bitu pomocniczego
      JU    omn;
      SET;
      R     L 4.7;
// Aby znalezc palete widmo
      A(;
      O     #i_Foto_Koniec_Wlot_1;
      O     #i_Foto_Koniec_Wlot_2;
      );
      AN    #Rel_Aktyw_z_Wlot_1;
      AN    #Rel_Aktyw_z_Wlot_2;
      AN    #Rel_Z_Nast_Aktywna;
      A(;
      L     #io_DW_Wartosc_Rej;
      L     0;
      ==D;
      );
      JCN   omn;
      SET;
      S     L 4.7;	//najstarszy bit (info o palecie)
      L     #Pom_LD4;
      T     #io_DW_Wartosc_Rej;
omn:  NOP   0;
NETWORK
TITLE =
//Przypisanie wartosci z pamieci podrecznej
//
      L     LW 0;
      T     #io_W_Pomoc;
      NOP   0;
END_FUNCTION

FUNCTION "Monitor_Bandy_+_Reczny" : VOID	// FC 315
//Funkcja na monitoruje przejezdzajacy miedzy bandami produkt
//Jezeli cos nie wyjdzie paleta widmo bierze wszystko na siebie
//
//
//0.7 - paleta obecna (nieuzywane)
//0.6 - kierunek spedycja (uzywane)
//0.5 - kierunek intro (uzywane)
//0.4 - wiazanie poprzeczne (uzywane)
//0.3 - wiazanie wzdluzne   (uzywane)
//0.2 - deklowanie (uzywane)
//0.1 - foliowanie (uzywane)
//0.0 - paleta obrabiana
//1.7 - rezerwa (nieuzywane)
//1.6 - rezerwa (nieuzywane)
//1.5 - rezerwa (nieuzywane)
//1.3 - rezerwa (nieuzywane)
//1.3 - info bit 3
//1.2 - info bit 2
//1.1 - info bit 1 
//1.0 - info bit 0
//
VERSION : 0.1
VAR_INPUT
  i_Auto_Reczny : BOOL ;	//1-Auto; 0-Reczny
  i_Foto_Tyl : BOOL ;
  i_Foto_Przod : BOOL ;
  i_Zabierz_Od_Pop : BOOL ;	//Sygnal zabierz od bandy poprzedniej
  i_Zabierz_Do_Nast : BOOL ;	//Sygnal zabierz do nastepnej
  i_Paleta_Dost_Od_Nast : BOOL ;
  i_Motor_Bandy_Tyl : BOOL ;
  i_Motor_Bandy_Przod : BOOL ;
  i_DW_Wartosc_Wej_Tyl : DINT ;	//Wartosc wejsciowa z poprzedniej bandy
  i_DW_Wartosc_Wej_Przod : DINT ;	//Wartosc wejsciowa z poprzedniej bandy
  Timmer_Kontroli : TIMER ;
END_VAR
VAR_IN_OUT
  io_DW_Wartosc_Rej : DINT ;	//Wartosc bierzaca rejestru
  io_W_Pomoc : WORD ;	//Slowo pomocnicze
END_VAR
VAR_TEMP
  Rel_Z_Pop_Aktywna : BOOL ;	//Relacja z banda poprzednia jest aktywna
  Rel_Z_Nast_Aktywna : BOOL ;	//Relacja z banda nastepna jest aktywan
  Help_Zbocze_1 : BOOL ;
  Help_Zbocze_2 : BOOL ;
  Help_Zbocze_3 : BOOL ;
  Help_Zbocze_4 : BOOL ;
  Help_Zbocze_5 : BOOL ;
  Pom_LB1 : BYTE ;
  Pom_LW2 : WORD ;
  Pom_LD4 : DINT ;
  Pom_LD8 : DINT ;
END_VAR
BEGIN
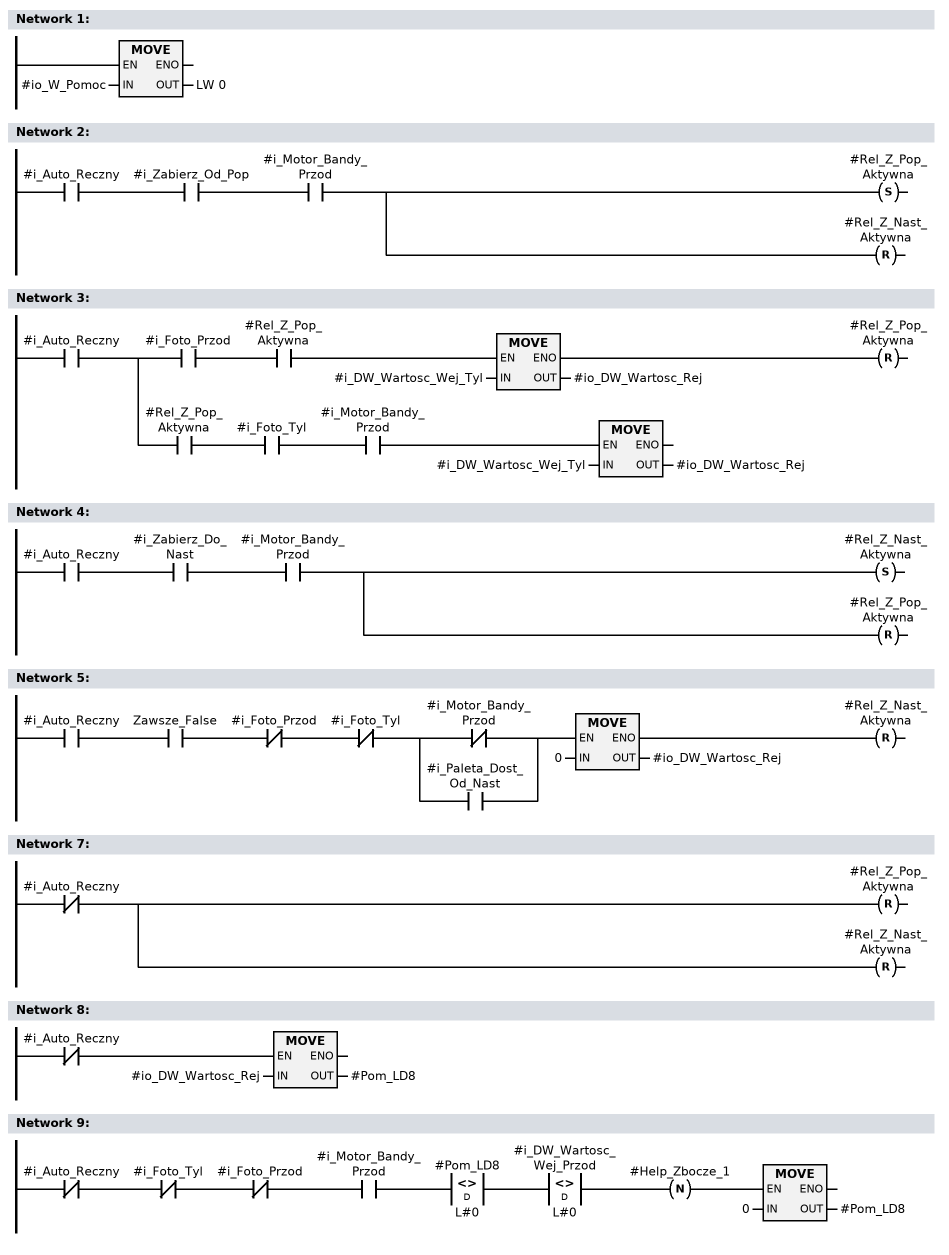
NETWORK
TITLE =
//Ten network celowo jest wolny
      L     #io_W_Pomoc;
      T     LW 0;
      NOP   0;
NETWORK
TITLE =
//Tryb Auto
//Pobranie wartosci
//
      A     #i_Auto_Reczny;
      A     #i_Zabierz_Od_Pop;
      A     #i_Motor_Bandy_Przod;
      S     #Rel_Z_Pop_Aktywna;
      R     #Rel_Z_Nast_Aktywna;
NETWORK
TITLE =
//Dojazd do fotokomorki i przepisanie wartosci.Informacja moze byc tez szybciej 
//przekazana (Gender potrzebuje szybciej)
      A     #i_Auto_Reczny;
      =     L 12.0;
      A     L 12.0;
      A     #i_Foto_Przod;
      A     #Rel_Z_Pop_Aktywna;
      JNB   _001;
      L     #i_DW_Wartosc_Wej_Tyl;
      T     #io_DW_Wartosc_Rej;
      SET;
      SAVE;
      CLR;
_001: A     BR;
      R     #Rel_Z_Pop_Aktywna;
      A     L 12.0;
      A     #Rel_Z_Pop_Aktywna;
      A     #i_Foto_Tyl;
      A     #i_Motor_Bandy_Przod;
      JNB   _002;
      L     #i_DW_Wartosc_Wej_Tyl;
      T     #io_DW_Wartosc_Rej;
_002: NOP   0;
NETWORK
TITLE =
//Relacja z nastepna banda
      A     #i_Auto_Reczny;
      A     #i_Zabierz_Do_Nast;
      A     #i_Motor_Bandy_Przod;
      S     #Rel_Z_Nast_Aktywna;
      R     #Rel_Z_Pop_Aktywna;
NETWORK
TITLE =
//Opuszczeni palety z bandy relacja przod
      A     #i_Auto_Reczny;
      A     "Zawsze_False";
      AN    #i_Foto_Przod;
      AN    #i_Foto_Tyl;
      A(;
      ON    #i_Motor_Bandy_Przod;
      O     #i_Paleta_Dost_Od_Nast;
      );
      JNB   _003;
      L     0;
      T     #io_DW_Wartosc_Rej;
      SET;
      SAVE;
      CLR;
_003: A     BR;
      R     #Rel_Z_Nast_Aktywna;
NETWORK
TITLE =
//Tryb Reczny
//Warunkiem prawidlowego dzialania trybu reczenego jest pokrycie zawsze co 
//najmniej jednej fotokomorki gdy jest produkt
//
//
NETWORK
TITLE =
//Zresetowanie relacji z automatyki
//
      AN    #i_Auto_Reczny;
      R     #Rel_Z_Pop_Aktywna;
      R     #Rel_Z_Nast_Aktywna;
NETWORK
TITLE =
//Trzeba sobie jakos radzic
      AN    #i_Auto_Reczny;
      JNB   _004;
      L     #io_DW_Wartosc_Rej;
      T     #Pom_LD8;
_004: NOP   0;
NETWORK
TITLE =
//Jazda do przodu na recznym.Bierzaca--->Nastepna
      AN    #i_Auto_Reczny;
      AN    #i_Foto_Tyl;
      AN    #i_Foto_Przod;
      A     #i_Motor_Bandy_Przod;
      A(;
      L     #Pom_LD8;
      L     L#0;
      <>D;
      );
      A(;
      L     #i_DW_Wartosc_Wej_Przod;
      L     L#0;
      <>D;
      );
      FN    #Help_Zbocze_1;
      JNB   _005;
      L     0;
      T     #Pom_LD8;
_005: NOP   0;
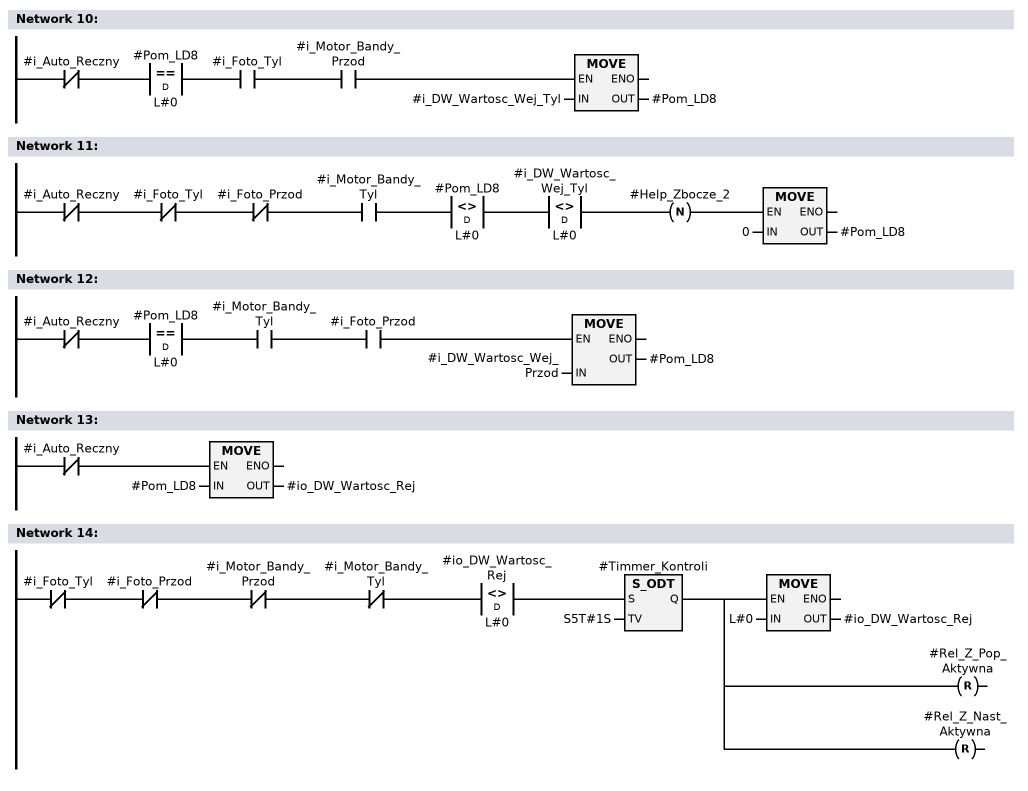
NETWORK
TITLE =
//Poprzednia wjezdza na bierzaca w trybie recznym. Poprzednia--->Bierzaca
      AN    #i_Auto_Reczny;
      A(;
      L     #Pom_LD8;
      L     L#0;
      ==D;
      );
      A     #i_Foto_Tyl;
      A     #i_Motor_Bandy_Przod;
      JNB   _006;
      L     #i_DW_Wartosc_Wej_Tyl;
      T     #Pom_LD8;
_006: NOP   0;
NETWORK
TITLE =
//Bierzaca wjezdza na bande porzedzajaca. Bierzaca--->Poprzednia
      AN    #i_Auto_Reczny;
      AN    #i_Foto_Tyl;
      AN    #i_Foto_Przod;
      A     #i_Motor_Bandy_Tyl;
      A(;
      L     #Pom_LD8;
      L     L#0;
      <>D;
      );
      A(;
      L     #i_DW_Wartosc_Wej_Tyl;
      L     L#0;
      <>D;
      );
      FN    #Help_Zbocze_2;
      JNB   _007;
      L     0;
      T     #Pom_LD8;
_007: NOP   0;
NETWORK
TITLE =
//Z Nastepnej wjezdza na bierzaca. Nastepna--->Bierzaca
      AN    #i_Auto_Reczny;
      A(;
      L     #Pom_LD8;
      L     L#0;
      ==D;
      );
      A     #i_Motor_Bandy_Tyl;
      A     #i_Foto_Przod;
      JNB   _008;
      L     #i_DW_Wartosc_Wej_Przod;
      T     #Pom_LD8;
_008: NOP   0;
NETWORK
TITLE =
//Przepisanie powrotne
      AN    #i_Auto_Reczny;
      JNB   _009;
      L     #Pom_LD8;
      T     #io_DW_Wartosc_Rej;
_009: NOP   0;
NETWORK
TITLE =
//Sprawdznie wszystkiego
//
      AN    #i_Foto_Tyl;
      AN    #i_Foto_Przod;
      AN    #i_Motor_Bandy_Przod;
      AN    #i_Motor_Bandy_Tyl;
      A(;
      L     #io_DW_Wartosc_Rej;
      L     L#0;
      <>D;
      );
      L     S5T#1S;
      SD    #Timmer_Kontroli;
      NOP   0;
      NOP   0;
      NOP   0;
      A     #Timmer_Kontroli;
      =     L 12.0;
      A     L 12.0;
      JNB   _00a;
      L     L#0;
      T     #io_DW_Wartosc_Rej;
_00a: NOP   0;
      A     L 12.0;
      BLD   102;
      R     #Rel_Z_Pop_Aktywna;
      A     L 12.0;
      BLD   102;
      R     #Rel_Z_Nast_Aktywna;
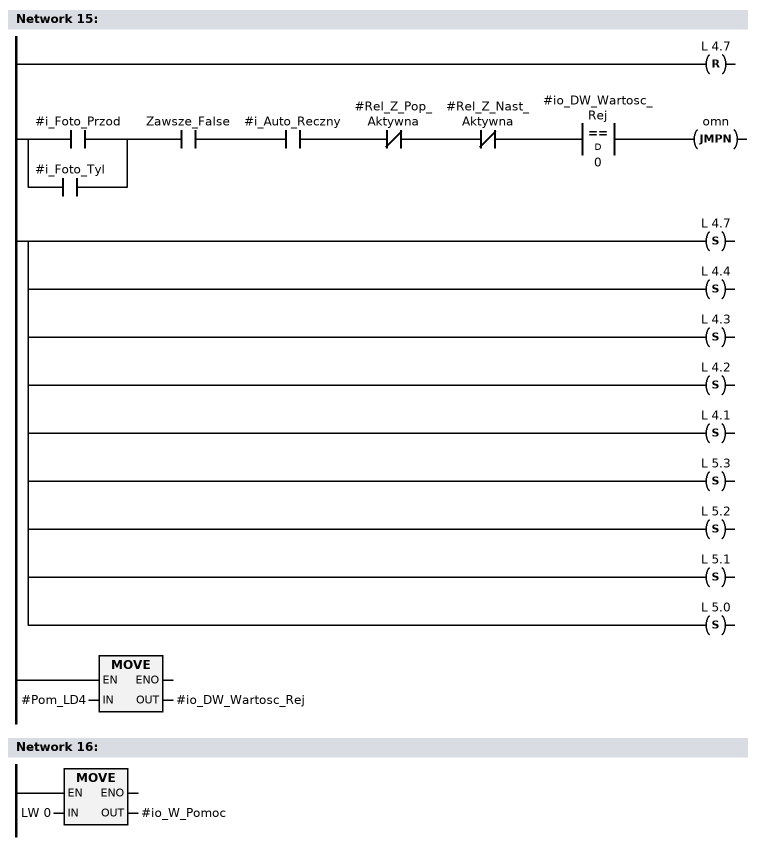
NETWORK
TITLE =
//0.7 - paleta obecna (nieuzywane)
//0.6 - kierunek spedycja (uzywane)
//0.5 - kierunek intro (uzywane)
//0.4 - wiazanie poprzeczne (uzywane)
//0.3 - wiazanie wzdluzne   (uzywane)
//0.2 - deklowanie (uzywane)
//0.1 - foliowanie (uzywane)
//0.0 - paleta obrabiana
//1.7 - rezerwa (nieuzywane)
//1.6 - rezerwa (nieuzywane)
//1.5 - rezerwa (nieuzywane)
//1.3 - rezerwa (nieuzywane)
//1.3 - info bit 3
//1.2 - info bit 2
//1.1 - info bit 1 
//1.0 - info bit 0
//
//kasowanie bitu pomocniczego
      SET;
      R     L 4.7;
// Aby znalezc palete widmo
      O     #i_Foto_Przod;
      O     #i_Foto_Tyl;
      A     "Zawsze_False";
      A     #i_Auto_Reczny;
      AN    #Rel_Z_Pop_Aktywna;
      AN    #Rel_Z_Nast_Aktywna;
      A(;
      L     #io_DW_Wartosc_Rej;
      L     0;
      ==D;
      );
      JCN   omn;
      SET;
      S     L 4.7;	//najstarszy bit (info o palecie)
      S     L 4.4;	//pop
      S     L 4.3;	//wzd
      S     L 4.2;	//dek
      S     L 4.1;	//fol
//--Daj znaczniki ze to paleta widmo
      S     L 5.3;
      S     L 5.2;
      S     L 5.1;
      S     L 5.0;
      L     #Pom_LD4;
      T     #io_DW_Wartosc_Rej;
omn:  NOP   0;
NETWORK
TITLE =
//Przypisanie wartosci z pamieci podrecznej
//
      L     LW 0;
      T     #io_W_Pomoc;
      NOP   0;
END_FUNCTION

FUNCTION "Monitor_Palety" : VOID	// FC 316
VERSION : 0.1
VAR_INPUT
  Foto_Pozycji_Przod : BOOL ;
  Foto_Pozycji_Tyl : BOOL ;	//Opcjonalna fotokomorka
END_VAR
VAR_IN_OUT
  iod_Wartosc_Rejestru : DINT ;
END_VAR
VAR_TEMP
  Wartosc_Pomocnicz_0 : DINT ;
  Wartosc_Pomocnicz_1 : DINT ;
END_VAR
BEGIN
NETWORK
TITLE =
      L     #iod_Wartosc_Rejestru;
      T     #Wartosc_Pomocnicz_0;
      O     #Foto_Pozycji_Przod;
      O     #Foto_Pozycji_Tyl;
      JCN   et_1;
      SET;
      S     L 0.7;
et_1: NOP   0;
      AN    #Foto_Pozycji_Przod;
      AN    #Foto_Pozycji_Tyl;
      JCN   et_2;
      SET;
      R     L 0.7;
et_2: NOP   0;
      L     #Wartosc_Pomocnicz_0;
      T     #iod_Wartosc_Rejestru;
END_FUNCTION

FUNCTION "Monitor_Bandy_2" : VOID	// FC 317
//Funkcja na monitoruje przejezdzajacy miedzy bandami produkt
//Jezeli cos nie wyjdzie paleta widmo bierze wszystko na siebie
//
//
//0.7 - paleta obecna (nieuzywane)
//0.6 - kierunek spedycja (uzywane)
//0.5 - kierunek intro (uzywane)
//0.4 - wiazanie poprzeczne (uzywane)
//0.3 - wiazanie wzdluzne   (uzywane)
//0.2 - deklowanie (uzywane)
//0.1 - foliowanie (uzywane)
//0.0 - paleta obrabiana
//1.7 - rezerwa (nieuzywane)
//1.6 - rezerwa (nieuzywane)
//1.5 - rezerwa (nieuzywane)
//1.3 - rezerwa (nieuzywane)
//1.3 - info bit 3
//1.2 - info bit 2
//1.1 - info bit 1 
//1.0 - info bit 0
//
VERSION : 0.1
VAR_INPUT
  i_Auto_Reczny : BOOL ;	//1-Auto; 0-Reczny
  i_Foto_Tyl : BOOL ;
  i_Foto_Przod : BOOL ;
  i_Zabierz_Od_Pop : BOOL ;	//Sygnal zabierz od bandy poprzedniej
  i_Zabierz_Do_Nast : BOOL ;	//Sygnal zabierz do nastepnej
  i_Paleta_Dost_Od_Nast : BOOL ;
  i_Motor_Bandy_Przod : BOOL ;
  i_DW_Wartosc_Wej_Tyl : DINT ;	//Wartosc wejsciowa z poprzedniej bandy
  i_DW_Wartosc_Wej_Przod : DINT ;
  Timmer_Kontroli : TIMER ;
END_VAR
VAR_IN_OUT
  io_DW_Wartosc_Rej : DINT ;	//Wartosc bierzaca rejestru
  io_W_Pomoc : WORD ;	//Slowo pomocnicze
END_VAR
VAR_TEMP
  Rel_Z_Pop_Aktywna : BOOL ;	//Relacja z banda poprzednia jest aktywna
  Rel_Z_Nast_Aktywna : BOOL ;	//Relacja z banda nastepna jest aktywan
  Help_Zbocze_1 : BOOL ;
  Help_Zbocze_2 : BOOL ;
  Help_Zbocze_3 : BOOL ;
  Help_Zbocze_4 : BOOL ;
  Help_Zbocze_5 : BOOL ;
  Pom_LB1 : BYTE ;
  Pom_LW2 : WORD ;
  Pom_LD4 : DINT ;
  Pom_LD8 : DINT ;
END_VAR
BEGIN
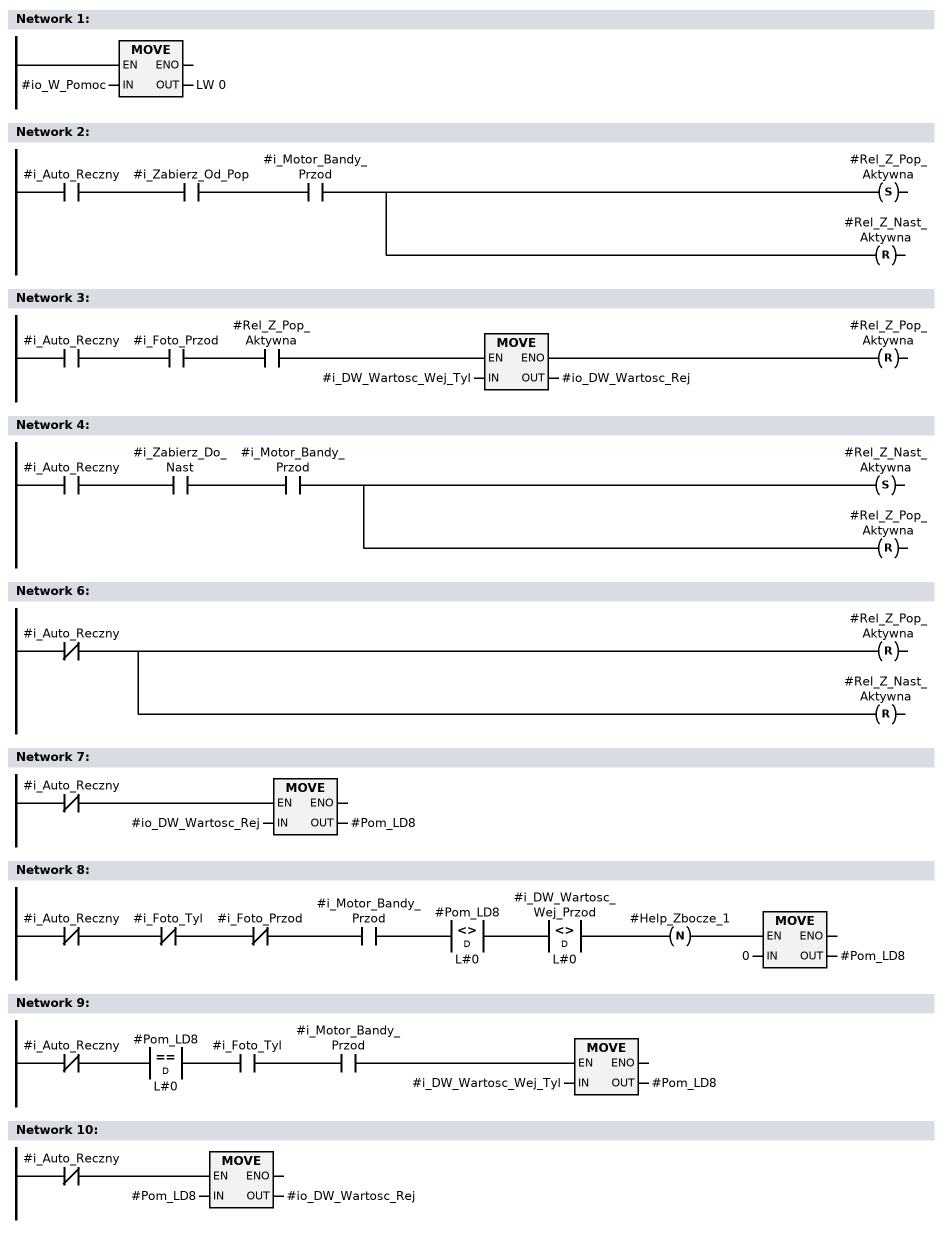
NETWORK
TITLE =
//Ten network celowo jest wolny
      L     #io_W_Pomoc;
      T     LW 0;
      NOP   0;
NETWORK
TITLE =
//Tryb Auto
//Pobranie wartosci
//
      A     #i_Auto_Reczny;
      A     #i_Zabierz_Od_Pop;
      A     #i_Motor_Bandy_Przod;
      S     #Rel_Z_Pop_Aktywna;
      R     #Rel_Z_Nast_Aktywna;
NETWORK
TITLE =
//Dojazd do fotokomorki i przepisanie wartosci.Informacja moze byc tez szybciej 
//przekazana (Gender potrzebuje szybciej)
      A     #i_Auto_Reczny;
      A     #i_Foto_Przod;
      A     #Rel_Z_Pop_Aktywna;
      JNB   _001;
      L     #i_DW_Wartosc_Wej_Tyl;
      T     #io_DW_Wartosc_Rej;
      SET;
      SAVE;
      CLR;
_001: A     BR;
      R     #Rel_Z_Pop_Aktywna;
NETWORK
TITLE =
//Relacja z nastepna banda
      A     #i_Auto_Reczny;
      A     #i_Zabierz_Do_Nast;
      A     #i_Motor_Bandy_Przod;
      S     #Rel_Z_Nast_Aktywna;
      R     #Rel_Z_Pop_Aktywna;
NETWORK
TITLE =
//Tryb Reczny
//Warunkiem prawidlowego dzialania trybu reczenego jest pokrycie zawsze co 
//najmniej jednej fotokomorki gdy jest produkt
//
//
NETWORK
TITLE =
//Zresetowanie relacji z automatyki
//
      AN    #i_Auto_Reczny;
      R     #Rel_Z_Pop_Aktywna;
      R     #Rel_Z_Nast_Aktywna;
NETWORK
TITLE =
//Trzeba sobie jakos radzic
      AN    #i_Auto_Reczny;
      JNB   _002;
      L     #io_DW_Wartosc_Rej;
      T     #Pom_LD8;
_002: NOP   0;
NETWORK
TITLE =
//Jazda do przodu na recznym.Bierzaca--->Nastepna
      AN    #i_Auto_Reczny;
      AN    #i_Foto_Tyl;
      AN    #i_Foto_Przod;
      A     #i_Motor_Bandy_Przod;
      A(;
      L     #Pom_LD8;
      L     L#0;
      <>D;
      );
      A(;
      L     #i_DW_Wartosc_Wej_Przod;
      L     L#0;
      <>D;
      );
      FN    #Help_Zbocze_1;
      JNB   _003;
      L     0;
      T     #Pom_LD8;
_003: NOP   0;
NETWORK
TITLE =
//Poprzednia wjezdza na bierzaca w trybie recznym. Poprzednia--->Bierzaca
      AN    #i_Auto_Reczny;
      A(;
      L     #Pom_LD8;
      L     L#0;
      ==D;
      );
      A     #i_Foto_Tyl;
      A     #i_Motor_Bandy_Przod;
      JNB   _004;
      L     #i_DW_Wartosc_Wej_Tyl;
      T     #Pom_LD8;
_004: NOP   0;
NETWORK
TITLE =
//Przepisanie powrotne
      AN    #i_Auto_Reczny;
      JNB   _005;
      L     #Pom_LD8;
      T     #io_DW_Wartosc_Rej;
_005: NOP   0;
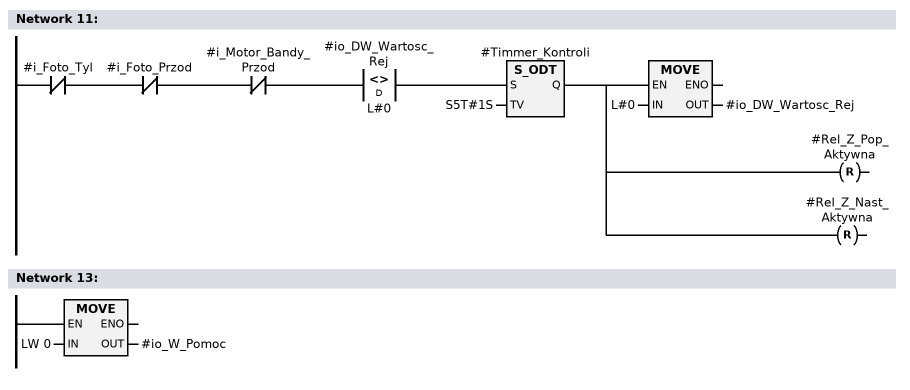
NETWORK
TITLE =
//Sprawdznie wszystkiego
//
      AN    #i_Foto_Tyl;
      AN    #i_Foto_Przod;
      AN    #i_Motor_Bandy_Przod;
      A(;
      L     #io_DW_Wartosc_Rej;
      L     L#0;
      <>D;
      );
      L     S5T#1S;
      SD    #Timmer_Kontroli;
      NOP   0;
      NOP   0;
      NOP   0;
      A     #Timmer_Kontroli;
      =     L 12.0;
      A     L 12.0;
      JNB   _006;
      L     L#0;
      T     #io_DW_Wartosc_Rej;
_006: NOP   0;
      A     L 12.0;
      BLD   102;
      R     #Rel_Z_Pop_Aktywna;
      A     L 12.0;
      BLD   102;
      R     #Rel_Z_Nast_Aktywna;
NETWORK
TITLE =
//0.7 - paleta obecna (nieuzywane)
//0.6 - kierunek spedycja (uzywane)
//0.5 - kierunek intro (uzywane)
//0.4 - wiazanie poprzeczne (uzywane)
//0.3 - wiazanie wzdluzne   (uzywane)
//0.2 - deklowanie (uzywane)
//0.1 - foliowanie (uzywane)
//0.0 - paleta obrabiana
//1.7 - rezerwa (nieuzywane)
//1.6 - rezerwa (nieuzywane)
//1.5 - rezerwa (nieuzywane)
//1.3 - rezerwa (nieuzywane)
//1.3 - info bit 3
//1.2 - info bit 2
//1.1 - info bit 1 
//1.0 - info bit 0
//
NETWORK
TITLE =
//Przypisanie wartosci z pamieci podrecznej
//
      L     LW 0;
      T     #io_W_Pomoc;
      NOP   0;
END_FUNCTION

FUNCTION "Monitor_Bandy_Obr_2" : VOID	// FC 318
//Funkcja na monitoruje przejezdzajacy miedzy bandami produkt
//Jezeli cos nie wyjdzie paleta widmo bierze wszystko na siebie
//
//
//0.7 - paleta obecna (nieuzywane)
//0.6 - kierunek spedycja (uzywane)
//0.5 - kierunek intro (uzywane)
//0.4 - wiazanie poprzeczne (uzywane)
//0.3 - wiazanie wzdluzne   (uzywane)
//0.2 - deklowanie (uzywane)
//0.1 - foliowanie (uzywane)
//0.0 - paleta obrabiana
//1.7 - rezerwa (nieuzywane)
//1.6 - rezerwa (nieuzywane)
//1.5 - rezerwa (nieuzywane)
//1.3 - rezerwa (nieuzywane)
//1.3 - info bit 3
//1.2 - info bit 2
//1.1 - info bit 1 
//1.0 - info bit 0
//
VERSION : 0.1
VAR_INPUT
  i_Foto_Tyl : BOOL ;
  i_Foto_Przod : BOOL ;
  i_Zabierz_Od_Wlot_1 : BOOL ;	//Sygnal zabierz od bandy poprzedniej
  i_Zabierz_Od_Wlot_2 : BOOL ;
  i_Zabierz_Do_Nast : BOOL ;	//Sygnal zabierz do nastepnej
  i_Paleta_Dost_Od_Nast : BOOL ;
  i_Motor_Przod_Wlot_1 : BOOL ;
  i_Motor_Przod_Wlot_2 : BOOL ;
  i_DW_Wart_Wej_Wlot_1 : DINT ;	//Wartosc wejsciowa z poprzedniej bandy
  i_DW_Wart_Wej_Wlot_2 : DINT ;
  i_DW_Wart_Wej_Przod : DINT ;
  Timmer_Kontroli : TIMER ;
END_VAR
VAR_IN_OUT
  io_DW_Wartosc_Rej : DINT ;	//Wartosc bierzaca rejestru
  io_W_Pomoc : WORD ;	//Slowo pomocnicze
END_VAR
VAR_TEMP
  Rel_Aktyw_z_Wlot_1 : BOOL ;	//Relacja z banda poprzednia jest aktywna
  Rel_Aktyw_z_Wlot_2 : BOOL ;
  Rel_Z_Nast_Aktywna : BOOL ;	//Relacja z banda nastepna jest aktywan
  Help_Zbocze_1 : BOOL ;
  Help_Zbocze_2 : BOOL ;
  Help_Zbocze_3 : BOOL ;
  Help_Zbocze_4 : BOOL ;
  Help_Zbocze_5 : BOOL ;
  Pom_LB1 : BYTE ;
  Pom_LW2 : WORD ;
  Pom_LD4 : DINT ;
  Pom_LD8 : DINT ;
END_VAR
BEGIN
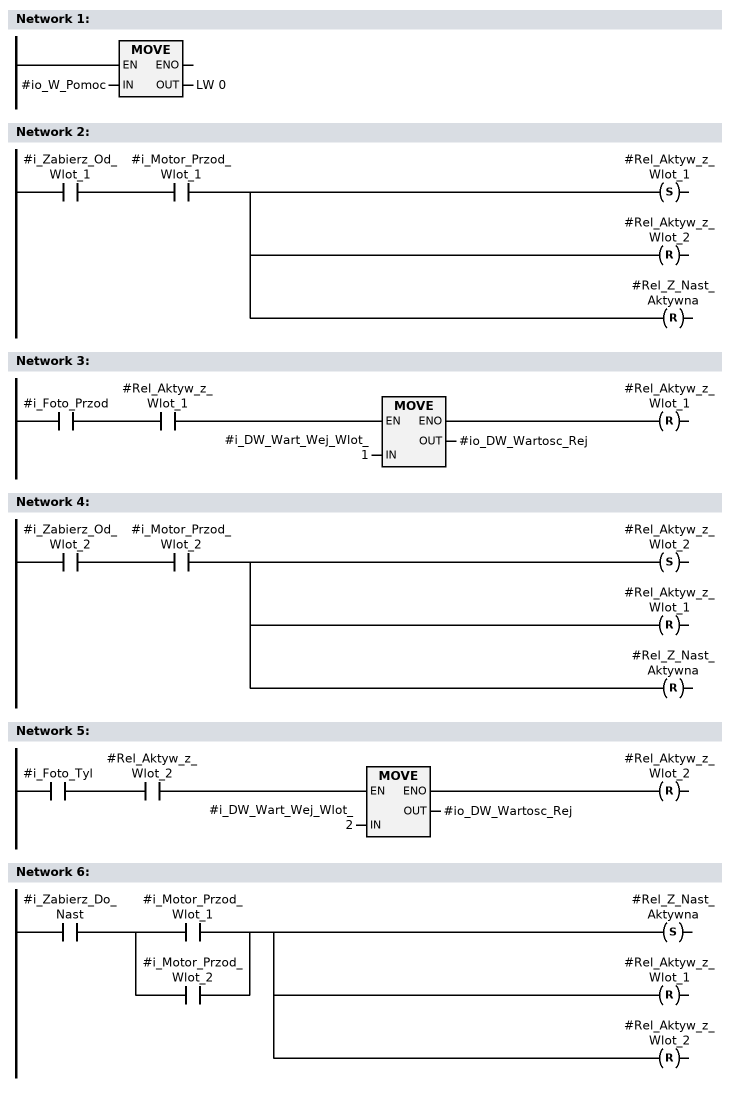
NETWORK
TITLE =
//Ten network celowo jest wolny
      L     #io_W_Pomoc;
      T     LW 0;
      NOP   0;
NETWORK
TITLE =
//Tryb Auto
//Pobranie wartosci
//
      A     #i_Zabierz_Od_Wlot_1;
      A     #i_Motor_Przod_Wlot_1;
      S     #Rel_Aktyw_z_Wlot_1;
      R     #Rel_Aktyw_z_Wlot_2;
      R     #Rel_Z_Nast_Aktywna;
NETWORK
TITLE =
//Dojazd do fotokomorki i przepisanie wartosci.Informacja moze byc tez szybciej 
//przekazana (Gender potrzebuje szybciej)
      A     #i_Foto_Przod;
      A     #Rel_Aktyw_z_Wlot_1;
      JNB   _001;
      L     #i_DW_Wart_Wej_Wlot_1;
      T     #io_DW_Wartosc_Rej;
      SET;
      SAVE;
      CLR;
_001: A     BR;
      R     #Rel_Aktyw_z_Wlot_1;
NETWORK
TITLE =
//Relacja z wlotem 2
//
      A     #i_Zabierz_Od_Wlot_2;
      A     #i_Motor_Przod_Wlot_2;
      S     #Rel_Aktyw_z_Wlot_2;
      R     #Rel_Aktyw_z_Wlot_1;
      R     #Rel_Z_Nast_Aktywna;
NETWORK
TITLE =
//Dojazd od strony bandy bocznej wtedy to foto tyl (foto_1) jest fotokomorka 
//tylna
      A     #i_Foto_Tyl;
      A     #Rel_Aktyw_z_Wlot_2;
      JNB   _002;
      L     #i_DW_Wart_Wej_Wlot_2;
      T     #io_DW_Wartosc_Rej;
      SET;
      SAVE;
      CLR;
_002: A     BR;
      R     #Rel_Aktyw_z_Wlot_2;
NETWORK
TITLE =
//Relacja z nastepna banda
      A     #i_Zabierz_Do_Nast;
      A(;
      O     #i_Motor_Przod_Wlot_1;
      O     #i_Motor_Przod_Wlot_2;
      );
      S     #Rel_Z_Nast_Aktywna;
      R     #Rel_Aktyw_z_Wlot_1;
      R     #Rel_Aktyw_z_Wlot_2;
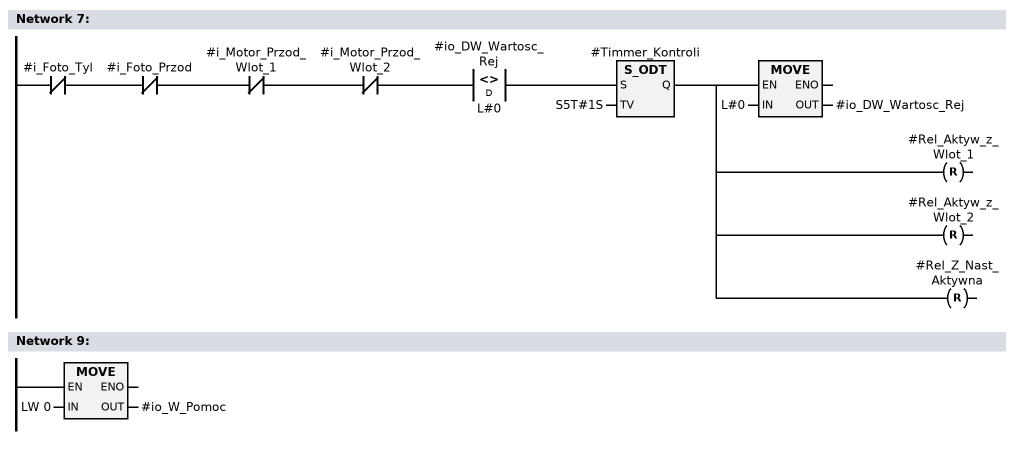
NETWORK
TITLE =
//Sprawdznie wszystkiego
//
      AN    #i_Foto_Tyl;
      AN    #i_Foto_Przod;
      AN    #i_Motor_Przod_Wlot_1;
      AN    #i_Motor_Przod_Wlot_2;
      A(;
      L     #io_DW_Wartosc_Rej;
      L     L#0;
      <>D;
      );
      L     S5T#1S;
      SD    #Timmer_Kontroli;
      NOP   0;
      NOP   0;
      NOP   0;
      A     #Timmer_Kontroli;
      =     L 12.0;
      A     L 12.0;
      JNB   _003;
      L     L#0;
      T     #io_DW_Wartosc_Rej;
_003: NOP   0;
      A     L 12.0;
      BLD   102;
      R     #Rel_Aktyw_z_Wlot_1;
      A     L 12.0;
      BLD   102;
      R     #Rel_Aktyw_z_Wlot_2;
      A     L 12.0;
      BLD   102;
      R     #Rel_Z_Nast_Aktywna;
NETWORK
TITLE =
//0.7 - paleta obecna (nieuzywane)
//0.6 - kierunek spedycja (uzywane)
//0.5 - kierunek intro (uzywane)
//0.4 - wiazanie poprzeczne (uzywane)
//0.3 - wiazanie wzdluzne   (uzywane)
//0.2 - deklowanie (uzywane)
//0.1 - foliowanie (uzywane)
//0.0 - paleta obrabiana
//1.7 - rezerwa (nieuzywane)
//1.6 - rezerwa (nieuzywane)
//1.5 - rezerwa (nieuzywane)
//1.3 - rezerwa (nieuzywane)
//1.3 - info bit 3
//1.2 - info bit 2
//1.1 - info bit 1 
//1.0 - info bit 0
//
NETWORK
TITLE =
//Przypisanie wartosci z pamieci podrecznej
//
      L     LW 0;
      T     #io_W_Pomoc;
      NOP   0;
END_FUNCTION

FUNCTION "Dekoduj_Maske" : VOID	// FC 320
//0.7 - paleta obecna (nieuzywane)
//0.6 - kierunek spedycja (uzywane)
//0.5 - kierunek intro (uzywane)
//0.4 - wiazanie poprzeczne (uzywane)
//0.3 - wiazanie wzdluzne   (uzywane)
//0.2 - deklowanie (uzywane)
//0.1 - foliowanie (uzywane)
//0.0 - paleta obrabiana
//1.7 - rezerwa (nieuzywane)
//1.6 - rezerwa (nieuzywane)
//1.5 - rezerwa (nieuzywane)
//1.3 - rezerwa (nieuzywane)
//1.3 - info bit 3
//1.2 - info bit 2
//1.1 - info bit 1 
//1.0 - info bit 0
//
VERSION : 0.1
VAR_INPUT
  Wartosc_Elementu : DINT ;
END_VAR
VAR_OUTPUT
  o_Paleta_Obecna : BOOL ;	//0.7
  o_Kierunek_Spedycja : BOOL ;	//0.6
  o_Kierunek_Intro : BOOL ;	//0.5
  o_Wizanie_Poprzeczne : BOOL ;	//0.4
  o_Wiazanie_Wzdluzne : BOOL ;	//0.3
  o_Deklowanie : BOOL ;	//0.2
  o_Foliowanie : BOOL ;	//0.1
  o_Paleta_Obrabiana : BOOL ;	//0.0
  o_Rezerwa_1_7 : BOOL ;	//1.7
  o_Rezerwa_1_6 : BOOL ;	//1.1
  o_Rezerwa_1_5 : BOOL ;	//1.2
  o_Rezerwa_1_4 : BOOL ;	//1.4
  o_Info_Bit_3 : BOOL ;	//1.3
  o_Info_Bit_2 : BOOL ;	//1.2
  o_Info_Bit_1 : BOOL ;	//1.1
  o_Info_Bit_0 : BOOL ;	//1.0
END_VAR
VAR_TEMP
  Edek_0 : DWORD ;
  Paleta_Obrabiana : BOOL ;	//0.0 - paleta_obrabiana
  Foliowanie : BOOL ;	//0.1
  Deklowanie : BOOL ;	//0.2
  Wiazanie_Wzdluzne : BOOL ;	//0.3
  Wizanie_Poprzeczne : BOOL ;	//0.4
  Kierunek_Intro : BOOL ;	//0.5
  Kierunek_Spedycja : BOOL ;	//0.6
  Paleta_Obecna : BOOL ;	//0.7
  Info_Bit_0 : BOOL ;	//1.0
  Info_Bit_1 : BOOL ;	//1.1
  Info_Bit_2 : BOOL ;	//1.2
  Info_Bit_3 : BOOL ;	//1.3
  Rezerwa_1_4 : BOOL ;	//1.4
  Rezerwa_1_5 : BOOL ;	//1.5
  Rezerwa_1_6 : BOOL ;	//1.6
  Rezerwa_1_7 : BOOL ;	//1.7
END_VAR
BEGIN
NETWORK
TITLE =
//ten network celowo jest wolny
NETWORK
TITLE =
//Zaladowanie maski
      L     #Wartosc_Elementu;
      T     LD 4;
NETWORK
TITLE =
//Wyluskanie zadan
      A     #Paleta_Obrabiana;
      =     #o_Paleta_Obrabiana;
//***
      A     #Foliowanie;
      =     #o_Foliowanie;
//***
      A     #Deklowanie;
      =     #o_Deklowanie;
//***
      A     #Wiazanie_Wzdluzne;
      =     #o_Wiazanie_Wzdluzne;
//***
      A     #Wizanie_Poprzeczne;
      =     #o_Wizanie_Poprzeczne;
//***
      A     #Kierunek_Intro;
      =     #o_Kierunek_Intro;
//***
      A     #Kierunek_Spedycja;
      =     #o_Kierunek_Spedycja;
//***
      A     #Paleta_Obecna;
      =     #o_Paleta_Obecna;
//***
      A     #Info_Bit_0;
      =     #o_Info_Bit_0;
//***
      A     #Info_Bit_1;
      =     #o_Info_Bit_1;
//***
      A     #Info_Bit_2;
      =     #o_Info_Bit_2;
//***
      A     #Info_Bit_3;
      =     #o_Info_Bit_3;
//***
      A     #Rezerwa_1_4;
      =     #o_Rezerwa_1_4;
//***
      A     #Rezerwa_1_5;
      =     #o_Rezerwa_1_5;
//***
      A     #Rezerwa_1_6;
      =     #o_Rezerwa_1_6;
//***
      A     #Rezerwa_1_7;
      =     #o_Rezerwa_1_7;
END_FUNCTION

FUNCTION "Nadpisz_Maske" : VOID	// FC 321
//Funkcja nadpisuje maske (bajt 2 i 3 ) informujac co dane stanowisko pracy 
//wykonalo
//
//0.7 - paleta obecna (nieuzywane)
//0.6 - kierunek spedycja (uzywane)
//0.5 - kierunek intro (uzywane)
//0.4 - wiazanie poprzeczne (uzywane)
//0.3 - wiazanie wzdluzne   (uzywane)
//0.2 - deklowanie (uzywane)
//0.1 - foliowanie (uzywane)
//0.0 - paleta obrabiana
//1.7 - rezerwa (nieuzywane)
//1.6 - rezerwa (nieuzywane)
//1.5 - rezerwa (nieuzywane)
//1.3 - rezerwa (nieuzywane)
//1.3 - info bit 3
//1.2 - info bit 2
//1.1 - info bit 1 
//1.0 - info bit 0
//
//
VERSION : 0.1
VAR_INPUT
  Nadpisz : BOOL ;
  i_Paleta_Obecna : BOOL ;	//0.7
  i_Kierunek_Spedycja : BOOL ;	//0.6
  i_Kierunek_Intro : BOOL ;	//0.5
  i_Wizanie_Poprzeczne : BOOL ;	//0.4
  i_Wiazanie_Wzdluzne : BOOL ;	//0.3
  i_Deklowanie : BOOL ;	//0.2
  i_Foliowanie : BOOL ;	//0.1
  i_Paleta_Obrabiana : BOOL ;	//0.0
  i_Rezerwa_1_7 : BOOL ;	//1.7
  i_Rezerwa_1_6 : BOOL ;	//1.1
  i_Rezerwa_1_5 : BOOL ;	//1.2
  i_Rezerwa_1_4 : BOOL ;	//1.4
  i_Info_Bit_3 : BOOL ;	//1.3
  i_Info_Bit_2 : BOOL ;	//1.2
  i_Info_Bit_1 : BOOL ;	//1.1
  i_Info_Bit_0 : BOOL ;	//1.0
END_VAR
VAR_IN_OUT
  Wartosc_Elementu : DINT ;
END_VAR
VAR_TEMP
  Edek_0 : DWORD ;
  INT_4_0 : INT ;
  Paleta_Obrabiana : BOOL ;	//0.0 - paleta_obrabiana
  Foliowanie : BOOL ;	//0.1
  Deklowanie : BOOL ;	//0.2
  Wiazanie_Wzdluzne : BOOL ;	//0.3
  Wizanie_Poprzeczne : BOOL ;	//0.4
  Kierunek_Intro : BOOL ;	//0.5
  Kierunek_Spedycja : BOOL ;	//0.6
  Paleta_Obecna : BOOL ;	//0.7
  Info_Bit_0 : BOOL ;	//1.0
  Info_Bit_1 : BOOL ;	//1.1
  Info_Bit_2 : BOOL ;	//1.2
  Info_Bit_3 : BOOL ;	//1.3
  Rezerwa_1_4 : BOOL ;	//1.4
  Rezerwa_1_5 : BOOL ;	//1.5
  Rezerwa_1_6 : BOOL ;	//1.6
  Rezerwa_1_7 : BOOL ;	//1.7
END_VAR
BEGIN
NETWORK
TITLE =
//ten network celowo jest wolny
NETWORK
TITLE =
//Zaladowanie maski
      L     #Wartosc_Elementu;
      T     LD 4;
NETWORK
TITLE =
//Wyluskanie zadan
      A     #Nadpisz;
      JCN   end;
      A     #i_Paleta_Obrabiana;
      =     #Paleta_Obrabiana;
//***
      A     #i_Foliowanie;
      =     #Foliowanie;
//***
      A     #i_Deklowanie;
      =     #Deklowanie;
//***
      A     #i_Wiazanie_Wzdluzne;
      =     #Wiazanie_Wzdluzne;
//***
      A     #i_Wizanie_Poprzeczne;
      =     #Wizanie_Poprzeczne;
//***
      A     #i_Kierunek_Intro;
      =     #Kierunek_Intro;
//***
      A     #i_Kierunek_Spedycja;
      =     #Kierunek_Spedycja;
//***
      A     #i_Paleta_Obecna;
      =     #Paleta_Obecna;
//***
      A     #i_Info_Bit_0;
      =     #Info_Bit_0;
//***
      A     #i_Info_Bit_1;
      =     #Info_Bit_1;
//***
      A     #i_Info_Bit_2;
      =     #Info_Bit_2;
//***
      A     #i_Info_Bit_3;
      =     #Info_Bit_3;
//***
      A     #i_Rezerwa_1_4;
      =     #Rezerwa_1_4;
//***
      A     #i_Rezerwa_1_5;
      =     #Rezerwa_1_5;
//***
      A     #i_Rezerwa_1_6;
      =     #Rezerwa_1_6;
//***
      A     #i_Rezerwa_1_7;
      =     #Rezerwa_1_7;
end:  L     LD 4;
      T     #Wartosc_Elementu;
END_FUNCTION

FUNCTION "Wirtualna_Foliarka" : VOID	// FC 330
VERSION : 0.1
BEGIN
NETWORK
TITLE =
//Ten Network celowo jest wolny
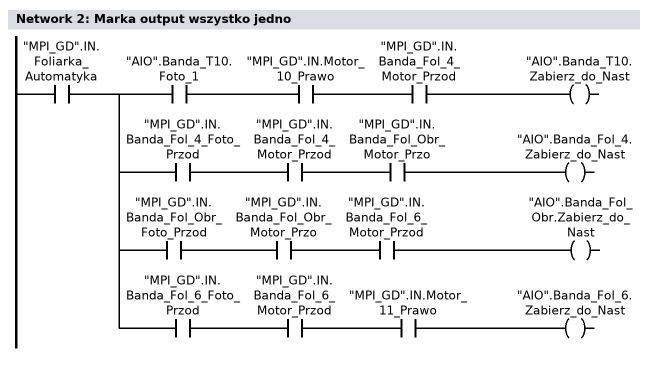
NETWORK
TITLE = Marka output wszystko jedno
//Przypisanie zabierz
//
      A     "MPI_GD".IN.Foliarka_Automatyka;
      =     L 0.0;
      A     L 0.0;
      A     "AIO".Banda_T10.Foto_1;
      A     "MPI_GD".IN.Motor_10_Prawo;
      A     "MPI_GD".IN.Banda_Fol_4_Motor_Przod;
      =     "AIO".Banda_T10.Zabierz_do_Nast;
      A     L 0.0;
      A     "MPI_GD".IN.Banda_Fol_4_Foto_Przod;
      A     "MPI_GD".IN.Banda_Fol_4_Motor_Przod;
      A     "MPI_GD".IN.Banda_Fol_Obr_Motor_Przo;
      =     "AIO".Banda_Fol_4.Zabierz_do_Nast;
      A     L 0.0;
      A     "MPI_GD".IN.Banda_Fol_Obr_Foto_Przod;
      A     "MPI_GD".IN.Banda_Fol_Obr_Motor_Przo;
      A     "MPI_GD".IN.Banda_Fol_6_Motor_Przod;
      =     "AIO".Banda_Fol_Obr.Zabierz_do_Nast;
      A     L 0.0;
      A     "MPI_GD".IN.Banda_Fol_6_Foto_Przod;
      A     "MPI_GD".IN.Banda_Fol_6_Motor_Przod;
      A     "MPI_GD".IN.Motor_11_Prawo;
      =     "AIO".Banda_Fol_6.Zabierz_do_Nast;
END_FUNCTION

DATA_BLOCK DB 4
VERSION : 0.0
"Czesc_Bindujaca"
BEGIN
END_DATA_BLOCK

DATA_BLOCK DB 5
VERSION : 0.0
"Czesc_Trasnportujaca"
BEGIN
END_DATA_BLOCK

DATA_BLOCK "AIO"	// DB 10
VERSION : 0.1
  STRUCT
   Banda_G1 : UDT 1;	//Temporary placeholder variable
   Banda_G2 : UDT 1;
   Banda_T3 : UDT 1;
   Banda_T4 : UDT 9;
   Banda_T5 : UDT 1;
   Banda_T6 : UDT 1;
   Banda_T7 : UDT 1;
   Banda_T8 : UDT 1;
   Banda_T9 : UDT 1;
   Banda_T10 : UDT 1;
   Banda_T11 : UDT 1;
   Banda_T12 : UDT 1;
   Banda_T13 : UDT 9;
   Banda_T14 : UDT 1;
   Obr_G15 : UDT 11;
   Czuj_G19_B : UDT 7;
   Czuj_G17_B : UDT 10;
   Obr_T18 : UDT 6;
   Czuj_T19 : UDT 7;
   Obr_T20 : UDT 6;
   Czuj_T21 : UDT 7;
   Czuj_T22 : UDT 8;
   Banda_G23 : UDT 1;
   Banda_G24 : UDT 1;
   Kurtyna_G25 : UDT 2;
   Kurtyna_G26 : UDT 2;
   ESTOP_T27 : UDT 3;
   ESTOP_T28 : UDT 3;
   ESTOP_T29 : UDT 3;
   ESTOP_T30 : UDT 3;
   ESTOP_TG31 : UDT 3;
   Rygiel_TG16 : UDT 2;
   Reset_TG17 : UDT 12;
   Reserwa_1 : UDT 1;
   Reserwa_2 : UDT 1;
   Banda_Fol_4 : UDT 1;
   Banda_Fol_Obr : UDT 1;
   Banda_Fol_6 : UDT 1;
  END_STRUCT ;	
BEGIN
END_DATA_BLOCK

DATA_BLOCK "Blok_Para"	// DB 12
VERSION : 0.1
  STRUCT
   Wiazanie_Poprzeczne : BOOL ;	//Wiaz wzdluz
   Wiazanie_Wzdluzne : BOOL ;
   Pozycjonowanie : BOOL ;
   Przelacz_Na_Auto : BOOL ;	//warunkowe przejscie na auto
   Start_Lini_z_OP : BOOL ;
   Stop_Lini_z_OP : BOOL ;
   Trigger_Wyjazd : BOOL ;	////wyjazd wtrybie auto
   Ser_Pokrycie_Foto : BOOL ;
   Pozycjon_Banda_Lewo : BOOL ;
   Pozycjon_Banda_Prawo : BOOL ;
   Pozycjon_Banda_Srodek : BOOL ;	//rozakaz pozycjonowana
   Banda_Poz_Lewa : BOOL ;
   Banda_Poz_Prawa : BOOL ;
   Banda_Poz_Srodek : BOOL ;
   Banda_Poz_Potw : BOOL ;
   Jedz_Na_0st : BOOL ;
   Jedz_Na_90st : BOOL ;
   Jedz_Na_180st : BOOL ;
   Jedz_Na_270st : BOOL ;
   Poz_0_st : BOOL ;
   Poz_90_st : BOOL ;
   Poz_180_st : BOOL ;
   Poz_270_st : BOOL ;
   Poz_Obr_Osiagnieta : BOOL ;
   Odblokuj_Rolki : BOOL ;
   Odblokuj_Obrotnice : BOOL ;
   Poz_Obr_Osiagnieta1 : BOOL ;
   Pozycja_Obrotnicy : INT ;
   Bin_Licznik : INT ;	//licznik bindownicy
   Rezerwa_Para : DWORD ;
   Krok_1 : BOOL ;
   krok_2 : BOOL ;
   krok_3 : BOOL ;
   krok_4 : BOOL ;
   krok_5 : BOOL ;
   krok_6 : BOOL ;
   krok_7 : BOOL ;
   krok_8 : BOOL ;
   krok_9 : BOOL ;
  END_STRUCT ;	
BEGIN
END_DATA_BLOCK

DATA_BLOCK "Blok_Bledow_Program"	// DB 13
VERSION : 0.1
  STRUCT
   Blad_Krok_1 : BOOL ;	//Blad kroku nr 1 (Przekrokczony czas jazdy  na zadana pozycje)
   Blad_Krok_2 : BOOL ;	//Blad kroku nr 2 (Przekrokczony czas szukania srodka palety)
   Blad_Krok_3 : BOOL ;	//Blad kroku nr 3 (Przekrokczony czas pozycjonowania palety lewo/prawo)
   Blad_Krok_4 : BOOL ;	//Blad kroku nr 4 (Przekrokczony czas strzalu bindownicy)
   Blad_Krok_5 : BOOL ;	//Blad kroku nr 6 (Przekrokczony czas czasu postoju)
   Blad_Krok_6 : BOOL ;	//Blad kroku nr 5 (Przekrokczony czas powrotu lewo/prawo)
   Blad_Krok_7 : BOOL ;	//Rezerwa
   Blad_Krok_8 : BOOL ;	//Rezerwa
   Blad_Krok_9 : BOOL ;	//Rezerwa
   Blad_Krok_10 : BOOL ;	//Rezerwa
  END_STRUCT ;	
BEGIN
END_DATA_BLOCK

DATA_BLOCK "Asi_input_Transport"	// DB 80
VERSION : 0.1
  STRUCT
   Adres_1_bit_0 : BOOL ;	//Temporary placeholder variable
   Adres_1_bit_1 : BOOL ;
   Adres_1_bit_2 : BOOL ;
   Adres_1_bit_3 : BOOL ;
   Adres_0_bit_0 : BOOL ;	//Temporary placeholder variable
   Adres_0_bit_1 : BOOL ;
   Adres_0_bit_2 : BOOL ;
   Adres_0_bit_3 : BOOL ;
   Adres_3_bit_0 : BOOL ;	//Temporary placeholder variable
   Adres_3_bit_1 : BOOL ;
   Adres_3_bit_2 : BOOL ;
   Adres_3_bit_3 : BOOL ;
   Adres_2_bit_0 : BOOL ;	//Temporary placeholder variable
   Adres_2_bit_1 : BOOL ;
   Adres_2_bit_2 : BOOL ;
   Adres_2_bit_3 : BOOL ;
   Adres_5_bit_0 : BOOL ;	//Temporary placeholder variable
   Adres_5_bit_1 : BOOL ;
   Adres_5_bit_2 : BOOL ;
   Adres_5_bit_3 : BOOL ;
   Adres_4_bit_0 : BOOL ;	//Temporary placeholder variable
   Adres_4_bit_1 : BOOL ;
   Adres_4_bit_2 : BOOL ;
   Adres_4_bit_3 : BOOL ;
   Adres_7_bit_0 : BOOL ;	//Temporary placeholder variable
   Adres_7_bit_1 : BOOL ;
   Adres_7_bit_2 : BOOL ;
   Adres_7_bit_3 : BOOL ;
   Adres_6_bit_0 : BOOL ;	//Temporary placeholder variable
   Adres_6_bit_1 : BOOL ;
   Adres_6_bit_2 : BOOL ;
   Adres_6_bit_3 : BOOL ;
   Adres_9_bit_0 : BOOL ;	//Temporary placeholder variable
   Adres_9_bit_1 : BOOL ;
   Adres_9_bit_2 : BOOL ;
   Adres_9_bit_3 : BOOL ;
   Adres_8_bit_0 : BOOL ;	//Temporary placeholder variable
   Adres_8_bit_1 : BOOL ;
   Adres_8_bit_2 : BOOL ;
   Adres_8_bit_3 : BOOL ;
   Adres_11_bit_0 : BOOL ;	//Temporary placeholder variable
   Adres_11_bit_1 : BOOL ;
   Adres_11_bit_2 : BOOL ;
   Adres_11_bit_3 : BOOL ;
   Adres_10_bit_0 : BOOL ;	//Temporary placeholder variable
   Adres_10_bit_1 : BOOL ;
   Adres_10_bit_2 : BOOL ;
   Adres_10_bit_3 : BOOL ;
   Adres_13_bit_0 : BOOL ;	//Temporary placeholder variable
   Adres_13_bit_1 : BOOL ;
   Adres_13_bit_2 : BOOL ;
   Adres_13_bit_3 : BOOL ;
   Adres_12_bit_0 : BOOL ;	//Temporary placeholder variable
   Adres_12_bit_1 : BOOL ;
   Adres_12_bit_2 : BOOL ;
   Adres_12_bit_3 : BOOL ;
   Adres_15_bit_0 : BOOL ;	//Temporary placeholder variable
   Adres_15_bit_1 : BOOL ;
   Adres_15_bit_2 : BOOL ;
   Adres_15_bit_3 : BOOL ;
   Adres_14_bit_0 : BOOL ;	//Temporary placeholder variable
   Adres_14_bit_1 : BOOL ;
   Adres_14_bit_2 : BOOL ;
   Adres_14_bit_3 : BOOL ;
   Adres_17_bit_0 : BOOL ;	//Temporary placeholder variable
   Adres_17_bit_1 : BOOL ;
   Adres_17_bit_2 : BOOL ;
   Adres_17_bit_3 : BOOL ;
   Adres_16_bit_0 : BOOL ;	//Temporary placeholder variable
   Adres_16_bit_1 : BOOL ;
   Adres_16_bit_2 : BOOL ;
   Adres_16_bit_3 : BOOL ;
   Adres_19_bit_0 : BOOL ;	//Temporary placeholder variable
   Adres_19_bit_1 : BOOL ;
   Adres_19_bit_2 : BOOL ;
   Adres_19_bit_3 : BOOL ;
   Adres_18_bit_0 : BOOL ;	//Temporary placeholder variable
   Adres_18_bit_1 : BOOL ;
   Adres_18_bit_2 : BOOL ;
   Adres_18_bit_3 : BOOL ;
   Adres_21_bit_0 : BOOL ;	//Temporary placeholder variable
   Adres_21_bit_1 : BOOL ;
   Adres_21_bit_2 : BOOL ;
   Adres_21_bit_3 : BOOL ;
   Adres_20_bit_0 : BOOL ;	//Temporary placeholder variable
   Adres_20_bit_1 : BOOL ;
   Adres_20_bit_2 : BOOL ;
   Adres_20_bit_3 : BOOL ;
   Adres_23_bit_0 : BOOL ;	//Temporary placeholder variable
   Adres_23_bit_1 : BOOL ;
   Adres_23_bit_2 : BOOL ;
   Adres_23_bit_3 : BOOL ;
   Adres_22_bit_0 : BOOL ;	//Temporary placeholder variable
   Adres_22_bit_1 : BOOL ;
   Adres_22_bit_2 : BOOL ;
   Adres_22_bit_3 : BOOL ;
   Adres_25_bit_0 : BOOL ;	//Temporary placeholder variable
   Adres_25_bit_1 : BOOL ;
   Adres_25_bit_2 : BOOL ;
   Adres_25_bit_3 : BOOL ;
   Adres_24_bit_0 : BOOL ;	//Temporary placeholder variable
   Adres_24_bit_1 : BOOL ;
   Adres_24_bit_2 : BOOL ;
   Adres_24_bit_3 : BOOL ;
   Adres_27_bit_0 : BOOL ;	//Temporary placeholder variable
   Adres_27_bit_1 : BOOL ;
   Adres_27_bit_2 : BOOL ;
   Adres_27_bit_3 : BOOL ;
   Adres_26_bit_0 : BOOL ;	//Temporary placeholder variable
   Adres_26_bit_1 : BOOL ;
   Adres_26_bit_2 : BOOL ;
   Adres_26_bit_3 : BOOL ;
   Adres_29_bit_0 : BOOL ;	//Temporary placeholder variable
   Adres_29_bit_1 : BOOL ;
   Adres_29_bit_2 : BOOL ;
   Adres_29_bit_3 : BOOL ;
   Adres_28_bit_0 : BOOL ;	//Temporary placeholder variable
   Adres_28_bit_1 : BOOL ;
   Adres_28_bit_2 : BOOL ;
   Adres_28_bit_3 : BOOL ;
   Adres_31_bit_0 : BOOL ;	//Temporary placeholder variable
   Adres_31_bit_1 : BOOL ;
   Adres_31_bit_2 : BOOL ;
   Adres_31_bit_3 : BOOL ;
   Adres_30_bit_0 : BOOL ;	//Temporary placeholder variable
   Adres_30_bit_1 : BOOL ;
   Adres_30_bit_2 : BOOL ;
   Adres_30_bit_3 : BOOL ;
   B_Adres_1_bit_0 : BOOL ;	//Temporary placeholder variable
   B_Adres_1_bit_1 : BOOL ;
   B_Adres_1_bit_2 : BOOL ;
   B_Adres_1_bit_3 : BOOL ;
   B_Adres_0_bit_0 : BOOL ;
   B_Adres_0_bit_1 : BOOL ;
   B_Adres_0_bit_2 : BOOL ;
   B_Adres_0_bit_3 : BOOL ;
   B_Adres_3_bit_0 : BOOL ;	//Temporary placeholder variable
   B_Adres_3_bit_1 : BOOL ;
   B_Adres_3_bit_2 : BOOL ;
   B_Adres_3_bit_3 : BOOL ;
   B_Adres_2_bit_0 : BOOL ;	//Temporary placeholder variable
   B_Adres_2_bit_1 : BOOL ;
   B_Adres_2_bit_2 : BOOL ;
   B_Adres_2_bit_3 : BOOL ;
   B_Adres_5_bit_0 : BOOL ;	//Temporary placeholder variable
   B_Adres_5_bit_1 : BOOL ;
   B_Adres_5_bit_2 : BOOL ;
   B_Adres_5_bit_3 : BOOL ;
   B_Adres_4_bit_0 : BOOL ;	//Temporary placeholder variable
   B_Adres_4_bit_1 : BOOL ;
   B_Adres_4_bit_2 : BOOL ;
   B_Adres_4_bit_3 : BOOL ;
   B_Adres_7_bit_0 : BOOL ;	//Temporary placeholder variable
   B_Adres_7_bit_1 : BOOL ;
   B_Adres_7_bit_2 : BOOL ;
   B_Adres_7_bit_3 : BOOL ;
   B_Adres_6_bit_0 : BOOL ;	//Temporary placeholder variable
   B_Adres_6_bit_1 : BOOL ;
   B_Adres_6_bit_2 : BOOL ;
   B_Adres_6_bit_3 : BOOL ;
   B_Adres_9_bit_0 : BOOL ;	//Temporary placeholder variable
   B_Adres_9_bit_1 : BOOL ;
   B_Adres_9_bit_2 : BOOL ;
   B_Adres_9_bit_3 : BOOL ;
   B_Adres_8_bit_0 : BOOL ;	//Temporary placeholder variable
   B_Adres_8_bit_1 : BOOL ;
   B_Adres_8_bit_2 : BOOL ;
   B_Adres_8_bit_3 : BOOL ;
   B_Adres_11_bit_0 : BOOL ;	//Temporary placeholder variable
   B_Adres_11_bit_1 : BOOL ;
   B_Adres_11_bit_2 : BOOL ;
   B_Adres_11_bit_3 : BOOL ;
   B_Adres_10_bit_0 : BOOL ;	//Temporary placeholder variable
   B_Adres_10_bit_1 : BOOL ;
   B_Adres_10_bit_2 : BOOL ;
   B_Adres_10_bit_3 : BOOL ;
   B_Adres_13_bit_0 : BOOL ;	//Temporary placeholder variable
   B_Adres_13_bit_1 : BOOL ;
   B_Adres_13_bit_2 : BOOL ;
   B_Adres_13_bit_3 : BOOL ;
   B_Adres_12_bit_0 : BOOL ;	//Temporary placeholder variable
   B_Adres_12_bit_1 : BOOL ;
   B_Adres_12_bit_2 : BOOL ;
   B_Adres_12_bit_3 : BOOL ;
   B_Adres_15_bit_0 : BOOL ;	//Temporary placeholder variable
   B_Adres_15_bit_1 : BOOL ;
   B_Adres_15_bit_2 : BOOL ;
   B_Adres_15_bit_3 : BOOL ;
   B_Adres_14_bit_0 : BOOL ;	//Temporary placeholder variable
   B_Adres_14_bit_1 : BOOL ;
   B_Adres_14_bit_2 : BOOL ;
   B_Adres_14_bit_3 : BOOL ;
   B_Adres_17_bit_0 : BOOL ;	//Temporary placeholder variable
   B_Adres_17_bit_1 : BOOL ;
   B_Adres_17_bit_2 : BOOL ;
   B_Adres_17_bit_3 : BOOL ;
   B_Adres_16_bit_0 : BOOL ;	//Temporary placeholder variable
   B_Adres_16_bit_1 : BOOL ;
   B_Adres_16_bit_2 : BOOL ;
   B_Adres_16_bit_3 : BOOL ;
   B_Adres_19_bit_0 : BOOL ;	//Temporary placeholder variable
   B_Adres_19_bit_1 : BOOL ;
   B_Adres_19_bit_2 : BOOL ;
   B_Adres_19_bit_3 : BOOL ;
   B_Adres_18_bit_0 : BOOL ;	//Temporary placeholder variable
   B_Adres_18_bit_1 : BOOL ;
   B_Adres_18_bit_2 : BOOL ;
   B_Adres_18_bit_3 : BOOL ;
   B_Adres_21_bit_0 : BOOL ;	//Temporary placeholder variable
   B_Adres_21_bit_1 : BOOL ;
   B_Adres_21_bit_2 : BOOL ;
   B_Adres_21_bit_3 : BOOL ;
   B_Adres_20_bit_0 : BOOL ;	//Temporary placeholder variable
   B_Adres_20_bit_1 : BOOL ;
   B_Adres_20_bit_2 : BOOL ;
   B_Adres_20_bit_3 : BOOL ;
   B_Adres_23_bit_0 : BOOL ;	//Temporary placeholder variable
   B_Adres_23_bit_1 : BOOL ;
   B_Adres_23_bit_2 : BOOL ;
   B_Adres_23_bit_3 : BOOL ;
   B_Adres_22_bit_0 : BOOL ;	//Temporary placeholder variable
   B_Adres_22_bit_1 : BOOL ;
   B_Adres_22_bit_2 : BOOL ;
   B_Adres_22_bit_3 : BOOL ;
   B_Adres_25_bit_0 : BOOL ;	//Temporary placeholder variable
   B_Adres_25_bit_1 : BOOL ;
   B_Adres_25_bit_2 : BOOL ;
   B_Adres_25_bit_3 : BOOL ;
   B_Adres_24_bit_0 : BOOL ;	//Temporary placeholder variable
   B_Adres_24_bit_1 : BOOL ;
   B_Adres_24_bit_2 : BOOL ;
   B_Adres_24_bit_3 : BOOL ;
   B_Adres_27_bit_0 : BOOL ;	//Temporary placeholder variable
   B_Adres_27_bit_1 : BOOL ;
   B_Adres_27_bit_2 : BOOL ;
   B_Adres_27_bit_3 : BOOL ;
   B_Adres_26_bit_0 : BOOL ;	//Temporary placeholder variable
   B_Adres_26_bit_1 : BOOL ;
   B_Adres_26_bit_2 : BOOL ;
   B_Adres_26_bit_3 : BOOL ;
   B_Adres_29_bit_0 : BOOL ;	//Temporary placeholder variable
   B_Adres_29_bit_1 : BOOL ;
   B_Adres_29_bit_2 : BOOL ;
   B_Adres_29_bit_3 : BOOL ;
   B_Adres_28_bit_0 : BOOL ;	//Temporary placeholder variable
   B_Adres_28_bit_1 : BOOL ;
   B_Adres_28_bit_2 : BOOL ;
   B_Adres_28_bit_3 : BOOL ;
   B_Adres_31_bit_0 : BOOL ;	//Temporary placeholder variable
   B_Adres_31_bit_1 : BOOL ;
   B_Adres_31_bit_2 : BOOL ;
   B_Adres_31_bit_3 : BOOL ;
   B_Adres_30_bit_0 : BOOL ;	//Temporary placeholder variable
   B_Adres_30_bit_1 : BOOL ;
   B_Adres_30_bit_2 : BOOL ;
   B_Adres_30_bit_3 : BOOL ;
  END_STRUCT ;	
BEGIN
END_DATA_BLOCK

DATA_BLOCK "Asi_output_Transport"	// DB 81
VERSION : 0.1
  STRUCT
   Adres_1_bit_0 : BOOL ;	//Temporary placeholder variable
   Adres_1_bit_1 : BOOL ;
   Adres_1_bit_2 : BOOL ;
   Adres_1_bit_3 : BOOL ;
   Adres_0_bit_0 : BOOL ;	//Temporary placeholder variable
   Adres_0_bit_1 : BOOL ;
   Adres_0_bit_2 : BOOL ;
   Adres_0_bit_3 : BOOL ;
   Adres_3_bit_0 : BOOL ;	//Temporary placeholder variable
   Adres_3_bit_1 : BOOL ;
   Adres_3_bit_2 : BOOL ;
   Adres_3_bit_3 : BOOL ;
   Adres_2_bit_0 : BOOL ;	//Temporary placeholder variable
   Adres_2_bit_1 : BOOL ;
   Adres_2_bit_2 : BOOL ;
   Adres_2_bit_3 : BOOL ;
   Adres_5_bit_0 : BOOL ;	//Temporary placeholder variable
   Adres_5_bit_1 : BOOL ;
   Adres_5_bit_2 : BOOL ;
   Adres_5_bit_3 : BOOL ;
   Adres_4_bit_0 : BOOL ;	//Temporary placeholder variable
   Adres_4_bit_1 : BOOL ;
   Adres_4_bit_2 : BOOL ;
   Adres_4_bit_3 : BOOL ;
   Adres_7_bit_0 : BOOL ;	//Temporary placeholder variable
   Adres_7_bit_1 : BOOL ;
   Adres_7_bit_2 : BOOL ;
   Adres_7_bit_3 : BOOL ;
   Adres_6_bit_0 : BOOL ;	//Temporary placeholder variable
   Adres_6_bit_1 : BOOL ;
   Adres_6_bit_2 : BOOL ;
   Adres_6_bit_3 : BOOL ;
   Adres_9_bit_0 : BOOL ;	//Temporary placeholder variable
   Adres_9_bit_1 : BOOL ;
   Adres_9_bit_2 : BOOL ;
   Adres_9_bit_3 : BOOL ;
   Adres_8_bit_0 : BOOL ;	//Temporary placeholder variable
   Adres_8_bit_1 : BOOL ;
   Adres_8_bit_2 : BOOL ;
   Adres_8_bit_3 : BOOL ;
   Adres_11_bit_0 : BOOL ;	//Temporary placeholder variable
   Adres_11_bit_1 : BOOL ;
   Adres_11_bit_2 : BOOL ;
   Adres_11_bit_3 : BOOL ;
   Adres_10_bit_0 : BOOL ;	//Temporary placeholder variable
   Adres_10_bit_1 : BOOL ;
   Adres_10_bit_2 : BOOL ;
   Adres_10_bit_3 : BOOL ;
   Adres_13_bit_0 : BOOL ;	//Temporary placeholder variable
   Adres_13_bit_1 : BOOL ;
   Adres_13_bit_2 : BOOL ;
   Adres_13_bit_3 : BOOL ;
   Adres_12_bit_0 : BOOL ;	//Temporary placeholder variable
   Adres_12_bit_1 : BOOL ;
   Adres_12_bit_2 : BOOL ;
   Adres_12_bit_3 : BOOL ;
   Adres_15_bit_0 : BOOL ;	//Temporary placeholder variable
   Adres_15_bit_1 : BOOL ;
   Adres_15_bit_2 : BOOL ;
   Adres_15_bit_3 : BOOL ;
   Adres_14_bit_0 : BOOL ;	//Temporary placeholder variable
   Adres_14_bit_1 : BOOL ;
   Adres_14_bit_2 : BOOL ;
   Adres_14_bit_3 : BOOL ;
   Adres_17_bit_0 : BOOL ;	//Temporary placeholder variable
   Adres_17_bit_1 : BOOL ;
   Adres_17_bit_2 : BOOL ;
   Adres_17_bit_3 : BOOL ;
   Adres_16_bit_0 : BOOL ;	//Temporary placeholder variable
   Adres_16_bit_1 : BOOL ;
   Adres_16_bit_2 : BOOL ;
   Adres_16_bit_3 : BOOL ;
   Adres_19_bit_0 : BOOL ;	//Temporary placeholder variable
   Adres_19_bit_1 : BOOL ;
   Adres_19_bit_2 : BOOL ;
   Adres_19_bit_3 : BOOL ;
   Adres_18_bit_0 : BOOL ;	//Temporary placeholder variable
   Adres_18_bit_1 : BOOL ;
   Adres_18_bit_2 : BOOL ;
   Adres_18_bit_3 : BOOL ;
   Adres_21_bit_0 : BOOL ;	//Temporary placeholder variable
   Adres_21_bit_1 : BOOL ;
   Adres_21_bit_2 : BOOL ;
   Adres_21_bit_3 : BOOL ;
   Adres_20_bit_0 : BOOL ;	//Temporary placeholder variable
   Adres_20_bit_1 : BOOL ;
   Adres_20_bit_2 : BOOL ;
   Adres_20_bit_3 : BOOL ;
   Adres_23_bit_0 : BOOL ;	//Temporary placeholder variable
   Adres_23_bit_1 : BOOL ;
   Adres_23_bit_2 : BOOL ;
   Adres_23_bit_3 : BOOL ;
   Adres_22_bit_0 : BOOL ;	//Temporary placeholder variable
   Adres_22_bit_1 : BOOL ;
   Adres_22_bit_2 : BOOL ;
   Adres_22_bit_3 : BOOL ;
   Adres_25_bit_0 : BOOL ;	//Temporary placeholder variable
   Adres_25_bit_1 : BOOL ;
   Adres_25_bit_2 : BOOL ;
   Adres_25_bit_3 : BOOL ;
   Adres_24_bit_0 : BOOL ;	//Temporary placeholder variable
   Adres_24_bit_1 : BOOL ;
   Adres_24_bit_2 : BOOL ;
   Adres_24_bit_3 : BOOL ;
   Adres_27_bit_0 : BOOL ;	//Temporary placeholder variable
   Adres_27_bit_1 : BOOL ;
   Adres_27_bit_2 : BOOL ;
   Adres_27_bit_3 : BOOL ;
   Adres_26_bit_0 : BOOL ;	//Temporary placeholder variable
   Adres_26_bit_1 : BOOL ;
   Adres_26_bit_2 : BOOL ;
   Adres_26_bit_3 : BOOL ;
   Adres_29_bit_0 : BOOL ;	//Temporary placeholder variable
   Adres_29_bit_1 : BOOL ;
   Adres_29_bit_2 : BOOL ;
   Adres_29_bit_3 : BOOL ;
   Adres_28_bit_0 : BOOL ;	//Temporary placeholder variable
   Adres_28_bit_1 : BOOL ;
   Adres_28_bit_2 : BOOL ;
   Adres_28_bit_3 : BOOL ;
   Adres_31_bit_0 : BOOL ;	//Temporary placeholder variable
   Adres_31_bit_1 : BOOL ;
   Adres_31_bit_2 : BOOL ;
   Adres_31_bit_3 : BOOL ;
   Adres_30_bit_0 : BOOL ;	//Temporary placeholder variable
   Adres_30_bit_1 : BOOL ;
   Adres_30_bit_2 : BOOL ;
   Adres_30_bit_3 : BOOL ;
   B_Adres_1_bit_0 : BOOL ;	//Temporary placeholder variable
   B_Adres_1_bit_1 : BOOL ;
   B_Adres_1_bit_2 : BOOL ;
   B_Adres_1_bit_3 : BOOL ;
   B_Adres_0_bit_0 : BOOL ;
   B_Adres_0_bit_1 : BOOL ;
   B_Adres_0_bit_2 : BOOL ;
   B_Adres_0_bit_3 : BOOL ;
   B_Adres_3_bit_0 : BOOL ;	//Temporary placeholder variable
   B_Adres_3_bit_1 : BOOL ;
   B_Adres_3_bit_2 : BOOL ;
   B_Adres_3_bit_3 : BOOL ;
   B_Adres_2_bit_0 : BOOL ;	//Temporary placeholder variable
   B_Adres_2_bit_1 : BOOL ;
   B_Adres_2_bit_2 : BOOL ;
   B_Adres_2_bit_3 : BOOL ;
   B_Adres_5_bit_0 : BOOL ;	//Temporary placeholder variable
   B_Adres_5_bit_1 : BOOL ;
   B_Adres_5_bit_2 : BOOL ;
   B_Adres_5_bit_3 : BOOL ;
   B_Adres_4_bit_0 : BOOL ;	//Temporary placeholder variable
   B_Adres_4_bit_1 : BOOL ;
   B_Adres_4_bit_2 : BOOL ;
   B_Adres_4_bit_3 : BOOL ;
   B_Adres_7_bit_0 : BOOL ;	//Temporary placeholder variable
   B_Adres_7_bit_1 : BOOL ;
   B_Adres_7_bit_2 : BOOL ;
   B_Adres_7_bit_3 : BOOL ;
   B_Adres_6_bit_0 : BOOL ;	//Temporary placeholder variable
   B_Adres_6_bit_1 : BOOL ;
   B_Adres_6_bit_2 : BOOL ;
   B_Adres_6_bit_3 : BOOL ;
   B_Adres_9_bit_0 : BOOL ;	//Temporary placeholder variable
   B_Adres_9_bit_1 : BOOL ;
   B_Adres_9_bit_2 : BOOL ;
   B_Adres_9_bit_3 : BOOL ;
   B_Adres_8_bit_0 : BOOL ;	//Temporary placeholder variable
   B_Adres_8_bit_1 : BOOL ;
   B_Adres_8_bit_2 : BOOL ;
   B_Adres_8_bit_3 : BOOL ;
   B_Adres_11_bit_0 : BOOL ;	//Temporary placeholder variable
   B_Adres_11_bit_1 : BOOL ;
   B_Adres_11_bit_2 : BOOL ;
   B_Adres_11_bit_3 : BOOL ;
   B_Adres_10_bit_0 : BOOL ;	//Temporary placeholder variable
   B_Adres_10_bit_1 : BOOL ;
   B_Adres_10_bit_2 : BOOL ;
   B_Adres_10_bit_3 : BOOL ;
   B_Adres_13_bit_0 : BOOL ;	//Temporary placeholder variable
   B_Adres_13_bit_1 : BOOL ;
   B_Adres_13_bit_2 : BOOL ;
   B_Adres_13_bit_3 : BOOL ;
   B_Adres_12_bit_0 : BOOL ;	//Temporary placeholder variable
   B_Adres_12_bit_1 : BOOL ;
   B_Adres_12_bit_2 : BOOL ;
   B_Adres_12_bit_3 : BOOL ;
   B_Adres_15_bit_0 : BOOL ;	//Temporary placeholder variable
   B_Adres_15_bit_1 : BOOL ;
   B_Adres_15_bit_2 : BOOL ;
   B_Adres_15_bit_3 : BOOL ;
   B_Adres_14_bit_0 : BOOL ;	//Temporary placeholder variable
   B_Adres_14_bit_1 : BOOL ;
   B_Adres_14_bit_2 : BOOL ;
   B_Adres_14_bit_3 : BOOL ;
   B_Adres_17_bit_0 : BOOL ;	//Temporary placeholder variable
   B_Adres_17_bit_1 : BOOL ;
   B_Adres_17_bit_2 : BOOL ;
   B_Adres_17_bit_3 : BOOL ;
   B_Adres_16_bit_0 : BOOL ;	//Temporary placeholder variable
   B_Adres_16_bit_1 : BOOL ;
   B_Adres_16_bit_2 : BOOL ;
   B_Adres_16_bit_3 : BOOL ;
   B_Adres_19_bit_0 : BOOL ;	//Temporary placeholder variable
   B_Adres_19_bit_1 : BOOL ;
   B_Adres_19_bit_2 : BOOL ;
   B_Adres_19_bit_3 : BOOL ;
   B_Adres_18_bit_0 : BOOL ;	//Temporary placeholder variable
   B_Adres_18_bit_1 : BOOL ;
   B_Adres_18_bit_2 : BOOL ;
   B_Adres_18_bit_3 : BOOL ;
   B_Adres_21_bit_0 : BOOL ;	//Temporary placeholder variable
   B_Adres_21_bit_1 : BOOL ;
   B_Adres_21_bit_2 : BOOL ;
   B_Adres_21_bit_3 : BOOL ;
   B_Adres_20_bit_0 : BOOL ;	//Temporary placeholder variable
   B_Adres_20_bit_1 : BOOL ;
   B_Adres_20_bit_2 : BOOL ;
   B_Adres_20_bit_3 : BOOL ;
   B_Adres_23_bit_0 : BOOL ;	//Temporary placeholder variable
   B_Adres_23_bit_1 : BOOL ;
   B_Adres_23_bit_2 : BOOL ;
   B_Adres_23_bit_3 : BOOL ;
   B_Adres_22_bit_0 : BOOL ;	//Temporary placeholder variable
   B_Adres_22_bit_1 : BOOL ;
   B_Adres_22_bit_2 : BOOL ;
   B_Adres_22_bit_3 : BOOL ;
   B_Adres_25_bit_0 : BOOL ;	//Temporary placeholder variable
   B_Adres_25_bit_1 : BOOL ;
   B_Adres_25_bit_2 : BOOL ;
   B_Adres_25_bit_3 : BOOL ;
   B_Adres_24_bit_0 : BOOL ;	//Temporary placeholder variable
   B_Adres_24_bit_1 : BOOL ;
   B_Adres_24_bit_2 : BOOL ;
   B_Adres_24_bit_3 : BOOL ;
   B_Adres_27_bit_0 : BOOL ;	//Temporary placeholder variable
   B_Adres_27_bit_1 : BOOL ;
   B_Adres_27_bit_2 : BOOL ;
   B_Adres_27_bit_3 : BOOL ;
   B_Adres_26_bit_0 : BOOL ;	//Temporary placeholder variable
   B_Adres_26_bit_1 : BOOL ;
   B_Adres_26_bit_2 : BOOL ;
   B_Adres_26_bit_3 : BOOL ;
   B_Adres_29_bit_0 : BOOL ;	//Temporary placeholder variable
   B_Adres_29_bit_1 : BOOL ;
   B_Adres_29_bit_2 : BOOL ;
   B_Adres_29_bit_3 : BOOL ;
   B_Adres_28_bit_0 : BOOL ;	//Temporary placeholder variable
   B_Adres_28_bit_1 : BOOL ;
   B_Adres_28_bit_2 : BOOL ;
   B_Adres_28_bit_3 : BOOL ;
   B_Adres_31_bit_0 : BOOL ;	//Temporary placeholder variable
   B_Adres_31_bit_1 : BOOL ;
   B_Adres_31_bit_2 : BOOL ;
   B_Adres_31_bit_3 : BOOL ;
   B_Adres_30_bit_0 : BOOL ;	//Temporary placeholder variable
   B_Adres_30_bit_1 : BOOL ;
   B_Adres_30_bit_2 : BOOL ;
   B_Adres_30_bit_3 : BOOL ;
  END_STRUCT ;	
BEGIN
END_DATA_BLOCK

DATA_BLOCK "Asi_Input_Gender"	// DB 82
VERSION : 0.1
  STRUCT
   Adres_1_bit_0 : BOOL ;	//Temporary placeholder variable
   Adres_1_bit_1 : BOOL ;
   Adres_1_bit_2 : BOOL ;
   Adres_1_bit_3 : BOOL ;
   Adres_0_bit_0 : BOOL ;	//Temporary placeholder variable
   Adres_0_bit_1 : BOOL ;
   Adres_0_bit_2 : BOOL ;
   Adres_0_bit_3 : BOOL ;
   Adres_3_bit_0 : BOOL ;	//Temporary placeholder variable
   Adres_3_bit_1 : BOOL ;
   Adres_3_bit_2 : BOOL ;
   Adres_3_bit_3 : BOOL ;
   Adres_2_bit_0 : BOOL ;	//Temporary placeholder variable
   Adres_2_bit_1 : BOOL ;
   Adres_2_bit_2 : BOOL ;
   Adres_2_bit_3 : BOOL ;
   Adres_5_bit_0 : BOOL ;	//Temporary placeholder variable
   Adres_5_bit_1 : BOOL ;
   Adres_5_bit_2 : BOOL ;
   Adres_5_bit_3 : BOOL ;
   Adres_4_bit_0 : BOOL ;	//Temporary placeholder variable
   Adres_4_bit_1 : BOOL ;
   Adres_4_bit_2 : BOOL ;
   Adres_4_bit_3 : BOOL ;
   Adres_7_bit_0 : BOOL ;	//Temporary placeholder variable
   Adres_7_bit_1 : BOOL ;
   Adres_7_bit_2 : BOOL ;
   Adres_7_bit_3 : BOOL ;
   Adres_6_bit_0 : BOOL ;	//Temporary placeholder variable
   Adres_6_bit_1 : BOOL ;
   Adres_6_bit_2 : BOOL ;
   Adres_6_bit_3 : BOOL ;
   Adres_9_bit_0 : BOOL ;	//Temporary placeholder variable
   Adres_9_bit_1 : BOOL ;
   Adres_9_bit_2 : BOOL ;
   Adres_9_bit_3 : BOOL ;
   Adres_8_bit_0 : BOOL ;	//Temporary placeholder variable
   Adres_8_bit_1 : BOOL ;
   Adres_8_bit_2 : BOOL ;
   Adres_8_bit_3 : BOOL ;
   Adres_11_bit_0 : BOOL ;	//Temporary placeholder variable
   Adres_11_bit_1 : BOOL ;
   Adres_11_bit_2 : BOOL ;
   Adres_11_bit_3 : BOOL ;
   Adres_10_bit_0 : BOOL ;	//Temporary placeholder variable
   Adres_10_bit_1 : BOOL ;
   Adres_10_bit_2 : BOOL ;
   Adres_10_bit_3 : BOOL ;
   Adres_13_bit_0 : BOOL ;	//Temporary placeholder variable
   Adres_13_bit_1 : BOOL ;
   Adres_13_bit_2 : BOOL ;
   Adres_13_bit_3 : BOOL ;
   Adres_12_bit_0 : BOOL ;	//Temporary placeholder variable
   Adres_12_bit_1 : BOOL ;
   Adres_12_bit_2 : BOOL ;
   Adres_12_bit_3 : BOOL ;
   Adres_15_bit_0 : BOOL ;	//Temporary placeholder variable
   Adres_15_bit_1 : BOOL ;
   Adres_15_bit_2 : BOOL ;
   Adres_15_bit_3 : BOOL ;
   Adres_14_bit_0 : BOOL ;	//Temporary placeholder variable
   Adres_14_bit_1 : BOOL ;
   Adres_14_bit_2 : BOOL ;
   Adres_14_bit_3 : BOOL ;
   Adres_17_bit_0 : BOOL ;	//Temporary placeholder variable
   Adres_17_bit_1 : BOOL ;
   Adres_17_bit_2 : BOOL ;
   Adres_17_bit_3 : BOOL ;
   Adres_16_bit_0 : BOOL ;	//Temporary placeholder variable
   Adres_16_bit_1 : BOOL ;
   Adres_16_bit_2 : BOOL ;
   Adres_16_bit_3 : BOOL ;
   Adres_19_bit_0 : BOOL ;	//Temporary placeholder variable
   Adres_19_bit_1 : BOOL ;
   Adres_19_bit_2 : BOOL ;
   Adres_19_bit_3 : BOOL ;
   Adres_18_bit_0 : BOOL ;	//Temporary placeholder variable
   Adres_18_bit_1 : BOOL ;
   Adres_18_bit_2 : BOOL ;
   Adres_18_bit_3 : BOOL ;
   Adres_21_bit_0 : BOOL ;	//Temporary placeholder variable
   Adres_21_bit_1 : BOOL ;
   Adres_21_bit_2 : BOOL ;
   Adres_21_bit_3 : BOOL ;
   Adres_20_bit_0 : BOOL ;	//Temporary placeholder variable
   Adres_20_bit_1 : BOOL ;
   Adres_20_bit_2 : BOOL ;
   Adres_20_bit_3 : BOOL ;
   Adres_23_bit_0 : BOOL ;	//Temporary placeholder variable
   Adres_23_bit_1 : BOOL ;
   Adres_23_bit_2 : BOOL ;
   Adres_23_bit_3 : BOOL ;
   Adres_22_bit_0 : BOOL ;	//Temporary placeholder variable
   Adres_22_bit_1 : BOOL ;
   Adres_22_bit_2 : BOOL ;
   Adres_22_bit_3 : BOOL ;
   Adres_25_bit_0 : BOOL ;	//Temporary placeholder variable
   Adres_25_bit_1 : BOOL ;
   Adres_25_bit_2 : BOOL ;
   Adres_25_bit_3 : BOOL ;
   Adres_24_bit_0 : BOOL ;	//Temporary placeholder variable
   Adres_24_bit_1 : BOOL ;
   Adres_24_bit_2 : BOOL ;
   Adres_24_bit_3 : BOOL ;
   Adres_27_bit_0 : BOOL ;	//Temporary placeholder variable
   Adres_27_bit_1 : BOOL ;
   Adres_27_bit_2 : BOOL ;
   Adres_27_bit_3 : BOOL ;
   Adres_26_bit_0 : BOOL ;	//Temporary placeholder variable
   Adres_26_bit_1 : BOOL ;
   Adres_26_bit_2 : BOOL ;
   Adres_26_bit_3 : BOOL ;
   Adres_29_bit_0 : BOOL ;	//Temporary placeholder variable
   Adres_29_bit_1 : BOOL ;
   Adres_29_bit_2 : BOOL ;
   Adres_29_bit_3 : BOOL ;
   Adres_28_bit_0 : BOOL ;	//Temporary placeholder variable
   Adres_28_bit_1 : BOOL ;
   Adres_28_bit_2 : BOOL ;
   Adres_28_bit_3 : BOOL ;
   Adres_31_bit_0 : BOOL ;	//Temporary placeholder variable
   Adres_31_bit_1 : BOOL ;
   Adres_31_bit_2 : BOOL ;
   Adres_31_bit_3 : BOOL ;
   Adres_30_bit_0 : BOOL ;	//Temporary placeholder variable
   Adres_30_bit_1 : BOOL ;
   Adres_30_bit_2 : BOOL ;
   Adres_30_bit_3 : BOOL ;
   B_Adres_1_bit_0 : BOOL ;	//Temporary placeholder variable
   B_Adres_1_bit_1 : BOOL ;
   B_Adres_1_bit_2 : BOOL ;
   B_Adres_1_bit_3 : BOOL ;
   B_Adres_0_bit_0 : BOOL ;
   B_Adres_0_bit_1 : BOOL ;
   B_Adres_0_bit_2 : BOOL ;
   B_Adres_0_bit_3 : BOOL ;
   B_Adres_3_bit_0 : BOOL ;	//Temporary placeholder variable
   B_Adres_3_bit_1 : BOOL ;
   B_Adres_3_bit_2 : BOOL ;
   B_Adres_3_bit_3 : BOOL ;
   B_Adres_2_bit_0 : BOOL ;	//Temporary placeholder variable
   B_Adres_2_bit_1 : BOOL ;
   B_Adres_2_bit_2 : BOOL ;
   B_Adres_2_bit_3 : BOOL ;
   B_Adres_5_bit_0 : BOOL ;	//Temporary placeholder variable
   B_Adres_5_bit_1 : BOOL ;
   B_Adres_5_bit_2 : BOOL ;
   B_Adres_5_bit_3 : BOOL ;
   B_Adres_4_bit_0 : BOOL ;	//Temporary placeholder variable
   B_Adres_4_bit_1 : BOOL ;
   B_Adres_4_bit_2 : BOOL ;
   B_Adres_4_bit_3 : BOOL ;
   B_Adres_7_bit_0 : BOOL ;	//Temporary placeholder variable
   B_Adres_7_bit_1 : BOOL ;
   B_Adres_7_bit_2 : BOOL ;
   B_Adres_7_bit_3 : BOOL ;
   B_Adres_6_bit_0 : BOOL ;	//Temporary placeholder variable
   B_Adres_6_bit_1 : BOOL ;
   B_Adres_6_bit_2 : BOOL ;
   B_Adres_6_bit_3 : BOOL ;
   B_Adres_9_bit_0 : BOOL ;	//Temporary placeholder variable
   B_Adres_9_bit_1 : BOOL ;
   B_Adres_9_bit_2 : BOOL ;
   B_Adres_9_bit_3 : BOOL ;
   B_Adres_8_bit_0 : BOOL ;	//Temporary placeholder variable
   B_Adres_8_bit_1 : BOOL ;
   B_Adres_8_bit_2 : BOOL ;
   B_Adres_8_bit_3 : BOOL ;
   B_Adres_11_bit_0 : BOOL ;	//Temporary placeholder variable
   B_Adres_11_bit_1 : BOOL ;
   B_Adres_11_bit_2 : BOOL ;
   B_Adres_11_bit_3 : BOOL ;
   B_Adres_10_bit_0 : BOOL ;	//Temporary placeholder variable
   B_Adres_10_bit_1 : BOOL ;
   B_Adres_10_bit_2 : BOOL ;
   B_Adres_10_bit_3 : BOOL ;
   B_Adres_13_bit_0 : BOOL ;	//Temporary placeholder variable
   B_Adres_13_bit_1 : BOOL ;
   B_Adres_13_bit_2 : BOOL ;
   B_Adres_13_bit_3 : BOOL ;
   B_Adres_12_bit_0 : BOOL ;	//Temporary placeholder variable
   B_Adres_12_bit_1 : BOOL ;
   B_Adres_12_bit_2 : BOOL ;
   B_Adres_12_bit_3 : BOOL ;
   B_Adres_15_bit_0 : BOOL ;	//Temporary placeholder variable
   B_Adres_15_bit_1 : BOOL ;
   B_Adres_15_bit_2 : BOOL ;
   B_Adres_15_bit_3 : BOOL ;
   B_Adres_14_bit_0 : BOOL ;	//Temporary placeholder variable
   B_Adres_14_bit_1 : BOOL ;
   B_Adres_14_bit_2 : BOOL ;
   B_Adres_14_bit_3 : BOOL ;
   B_Adres_17_bit_0 : BOOL ;	//Temporary placeholder variable
   B_Adres_17_bit_1 : BOOL ;
   B_Adres_17_bit_2 : BOOL ;
   B_Adres_17_bit_3 : BOOL ;
   B_Adres_16_bit_0 : BOOL ;	//Temporary placeholder variable
   B_Adres_16_bit_1 : BOOL ;
   B_Adres_16_bit_2 : BOOL ;
   B_Adres_16_bit_3 : BOOL ;
   B_Adres_19_bit_0 : BOOL ;	//Temporary placeholder variable
   B_Adres_19_bit_1 : BOOL ;
   B_Adres_19_bit_2 : BOOL ;
   B_Adres_19_bit_3 : BOOL ;
   B_Adres_18_bit_0 : BOOL ;	//Temporary placeholder variable
   B_Adres_18_bit_1 : BOOL ;
   B_Adres_18_bit_2 : BOOL ;
   B_Adres_18_bit_3 : BOOL ;
   B_Adres_21_bit_0 : BOOL ;	//Temporary placeholder variable
   B_Adres_21_bit_1 : BOOL ;
   B_Adres_21_bit_2 : BOOL ;
   B_Adres_21_bit_3 : BOOL ;
   B_Adres_20_bit_0 : BOOL ;	//Temporary placeholder variable
   B_Adres_20_bit_1 : BOOL ;
   B_Adres_20_bit_2 : BOOL ;
   B_Adres_20_bit_3 : BOOL ;
   B_Adres_23_bit_0 : BOOL ;	//Temporary placeholder variable
   B_Adres_23_bit_1 : BOOL ;
   B_Adres_23_bit_2 : BOOL ;
   B_Adres_23_bit_3 : BOOL ;
   B_Adres_22_bit_0 : BOOL ;	//Temporary placeholder variable
   B_Adres_22_bit_1 : BOOL ;
   B_Adres_22_bit_2 : BOOL ;
   B_Adres_22_bit_3 : BOOL ;
   B_Adres_25_bit_0 : BOOL ;	//Temporary placeholder variable
   B_Adres_25_bit_1 : BOOL ;
   B_Adres_25_bit_2 : BOOL ;
   B_Adres_25_bit_3 : BOOL ;
   B_Adres_24_bit_0 : BOOL ;	//Temporary placeholder variable
   B_Adres_24_bit_1 : BOOL ;
   B_Adres_24_bit_2 : BOOL ;
   B_Adres_24_bit_3 : BOOL ;
   B_Adres_27_bit_0 : BOOL ;	//Temporary placeholder variable
   B_Adres_27_bit_1 : BOOL ;
   B_Adres_27_bit_2 : BOOL ;
   B_Adres_27_bit_3 : BOOL ;
   B_Adres_26_bit_0 : BOOL ;	//Temporary placeholder variable
   B_Adres_26_bit_1 : BOOL ;
   B_Adres_26_bit_2 : BOOL ;
   B_Adres_26_bit_3 : BOOL ;
   B_Adres_29_bit_0 : BOOL ;	//Temporary placeholder variable
   B_Adres_29_bit_1 : BOOL ;
   B_Adres_29_bit_2 : BOOL ;
   B_Adres_29_bit_3 : BOOL ;
   B_Adres_28_bit_0 : BOOL ;	//Temporary placeholder variable
   B_Adres_28_bit_1 : BOOL ;
   B_Adres_28_bit_2 : BOOL ;
   B_Adres_28_bit_3 : BOOL ;
   B_Adres_31_bit_0 : BOOL ;	//Temporary placeholder variable
   B_Adres_31_bit_1 : BOOL ;
   B_Adres_31_bit_2 : BOOL ;
   B_Adres_31_bit_3 : BOOL ;
   B_Adres_30_bit_0 : BOOL ;	//Temporary placeholder variable
   B_Adres_30_bit_1 : BOOL ;
   B_Adres_30_bit_2 : BOOL ;
   B_Adres_30_bit_3 : BOOL ;
  END_STRUCT ;	
BEGIN
END_DATA_BLOCK

DATA_BLOCK "Asi_Output_Gender"	// DB 83
VERSION : 0.1
  STRUCT
   Adres_1_bit_0 : BOOL ;	//Temporary placeholder variable
   Adres_1_bit_1 : BOOL ;
   Adres_1_bit_2 : BOOL ;
   Adres_1_bit_3 : BOOL ;
   Adres_0_bit_0 : BOOL ;	//Temporary placeholder variable
   Adres_0_bit_1 : BOOL ;
   Adres_0_bit_2 : BOOL ;
   Adres_0_bit_3 : BOOL ;
   Adres_3_bit_0 : BOOL ;	//Temporary placeholder variable
   Adres_3_bit_1 : BOOL ;
   Adres_3_bit_2 : BOOL ;
   Adres_3_bit_3 : BOOL ;
   Adres_2_bit_0 : BOOL ;	//Temporary placeholder variable
   Adres_2_bit_1 : BOOL ;
   Adres_2_bit_2 : BOOL ;
   Adres_2_bit_3 : BOOL ;
   Adres_5_bit_0 : BOOL ;	//Temporary placeholder variable
   Adres_5_bit_1 : BOOL ;
   Adres_5_bit_2 : BOOL ;
   Adres_5_bit_3 : BOOL ;
   Adres_4_bit_0 : BOOL ;	//Temporary placeholder variable
   Adres_4_bit_1 : BOOL ;
   Adres_4_bit_2 : BOOL ;
   Adres_4_bit_3 : BOOL ;
   Adres_7_bit_0 : BOOL ;	//Temporary placeholder variable
   Adres_7_bit_1 : BOOL ;
   Adres_7_bit_2 : BOOL ;
   Adres_7_bit_3 : BOOL ;
   Adres_6_bit_0 : BOOL ;	//Temporary placeholder variable
   Adres_6_bit_1 : BOOL ;
   Adres_6_bit_2 : BOOL ;
   Adres_6_bit_3 : BOOL ;
   Adres_9_bit_0 : BOOL ;	//Temporary placeholder variable
   Adres_9_bit_1 : BOOL ;
   Adres_9_bit_2 : BOOL ;
   Adres_9_bit_3 : BOOL ;
   Adres_8_bit_0 : BOOL ;	//Temporary placeholder variable
   Adres_8_bit_1 : BOOL ;
   Adres_8_bit_2 : BOOL ;
   Adres_8_bit_3 : BOOL ;
   Adres_11_bit_0 : BOOL ;	//Temporary placeholder variable
   Adres_11_bit_1 : BOOL ;
   Adres_11_bit_2 : BOOL ;
   Adres_11_bit_3 : BOOL ;
   Adres_10_bit_0 : BOOL ;	//Temporary placeholder variable
   Adres_10_bit_1 : BOOL ;
   Adres_10_bit_2 : BOOL ;
   Adres_10_bit_3 : BOOL ;
   Adres_13_bit_0 : BOOL ;	//Temporary placeholder variable
   Adres_13_bit_1 : BOOL ;
   Adres_13_bit_2 : BOOL ;
   Adres_13_bit_3 : BOOL ;
   Adres_12_bit_0 : BOOL ;	//Temporary placeholder variable
   Adres_12_bit_1 : BOOL ;
   Adres_12_bit_2 : BOOL ;
   Adres_12_bit_3 : BOOL ;
   Adres_15_bit_0 : BOOL ;	//Temporary placeholder variable
   Adres_15_bit_1 : BOOL ;
   Adres_15_bit_2 : BOOL ;
   Adres_15_bit_3 : BOOL ;
   Adres_14_bit_0 : BOOL ;	//Temporary placeholder variable
   Adres_14_bit_1 : BOOL ;
   Adres_14_bit_2 : BOOL ;
   Adres_14_bit_3 : BOOL ;
   Adres_17_bit_0 : BOOL ;	//Temporary placeholder variable
   Adres_17_bit_1 : BOOL ;
   Adres_17_bit_2 : BOOL ;
   Adres_17_bit_3 : BOOL ;
   Adres_16_bit_0 : BOOL ;	//Temporary placeholder variable
   Adres_16_bit_1 : BOOL ;
   Adres_16_bit_2 : BOOL ;
   Adres_16_bit_3 : BOOL ;
   Adres_19_bit_0 : BOOL ;	//Temporary placeholder variable
   Adres_19_bit_1 : BOOL ;
   Adres_19_bit_2 : BOOL ;
   Adres_19_bit_3 : BOOL ;
   Adres_18_bit_0 : BOOL ;	//Temporary placeholder variable
   Adres_18_bit_1 : BOOL ;
   Adres_18_bit_2 : BOOL ;
   Adres_18_bit_3 : BOOL ;
   Adres_21_bit_0 : BOOL ;	//Temporary placeholder variable
   Adres_21_bit_1 : BOOL ;
   Adres_21_bit_2 : BOOL ;
   Adres_21_bit_3 : BOOL ;
   Adres_20_bit_0 : BOOL ;	//Temporary placeholder variable
   Adres_20_bit_1 : BOOL ;
   Adres_20_bit_2 : BOOL ;
   Adres_20_bit_3 : BOOL ;
   Adres_23_bit_0 : BOOL ;	//Temporary placeholder variable
   Adres_23_bit_1 : BOOL ;
   Adres_23_bit_2 : BOOL ;
   Adres_23_bit_3 : BOOL ;
   Adres_22_bit_0 : BOOL ;	//Temporary placeholder variable
   Adres_22_bit_1 : BOOL ;
   Adres_22_bit_2 : BOOL ;
   Adres_22_bit_3 : BOOL ;
   Adres_25_bit_0 : BOOL ;	//Temporary placeholder variable
   Adres_25_bit_1 : BOOL ;
   Adres_25_bit_2 : BOOL ;
   Adres_25_bit_3 : BOOL ;
   Adres_24_bit_0 : BOOL ;	//Temporary placeholder variable
   Adres_24_bit_1 : BOOL ;
   Adres_24_bit_2 : BOOL ;
   Adres_24_bit_3 : BOOL ;
   Adres_27_bit_0 : BOOL ;	//Temporary placeholder variable
   Adres_27_bit_1 : BOOL ;
   Adres_27_bit_2 : BOOL ;
   Adres_27_bit_3 : BOOL ;
   Adres_26_bit_0 : BOOL ;	//Temporary placeholder variable
   Adres_26_bit_1 : BOOL ;
   Adres_26_bit_2 : BOOL ;
   Adres_26_bit_3 : BOOL ;
   Adres_29_bit_0 : BOOL ;	//Temporary placeholder variable
   Adres_29_bit_1 : BOOL ;
   Adres_29_bit_2 : BOOL ;
   Adres_29_bit_3 : BOOL ;
   Adres_28_bit_0 : BOOL ;	//Temporary placeholder variable
   Adres_28_bit_1 : BOOL ;
   Adres_28_bit_2 : BOOL ;
   Adres_28_bit_3 : BOOL ;
   Adres_31_bit_0 : BOOL ;	//Temporary placeholder variable
   Adres_31_bit_1 : BOOL ;
   Adres_31_bit_2 : BOOL ;
   Adres_31_bit_3 : BOOL ;
   Adres_30_bit_0 : BOOL ;	//Temporary placeholder variable
   Adres_30_bit_1 : BOOL ;
   Adres_30_bit_2 : BOOL ;
   Adres_30_bit_3 : BOOL ;
   B_Adres_1_bit_0 : BOOL ;	//Temporary placeholder variable
   B_Adres_1_bit_1 : BOOL ;
   B_Adres_1_bit_2 : BOOL ;
   B_Adres_1_bit_3 : BOOL ;
   B_Adres_0_bit_0 : BOOL ;
   B_Adres_0_bit_1 : BOOL ;
   B_Adres_0_bit_2 : BOOL ;
   B_Adres_0_bit_3 : BOOL ;
   B_Adres_3_bit_0 : BOOL ;	//Temporary placeholder variable
   B_Adres_3_bit_1 : BOOL ;
   B_Adres_3_bit_2 : BOOL ;
   B_Adres_3_bit_3 : BOOL ;
   B_Adres_2_bit_0 : BOOL ;	//Temporary placeholder variable
   B_Adres_2_bit_1 : BOOL ;
   B_Adres_2_bit_2 : BOOL ;
   B_Adres_2_bit_3 : BOOL ;
   B_Adres_5_bit_0 : BOOL ;	//Temporary placeholder variable
   B_Adres_5_bit_1 : BOOL ;
   B_Adres_5_bit_2 : BOOL ;
   B_Adres_5_bit_3 : BOOL ;
   B_Adres_4_bit_0 : BOOL ;	//Temporary placeholder variable
   B_Adres_4_bit_1 : BOOL ;
   B_Adres_4_bit_2 : BOOL ;
   B_Adres_4_bit_3 : BOOL ;
   B_Adres_7_bit_0 : BOOL ;	//Temporary placeholder variable
   B_Adres_7_bit_1 : BOOL ;
   B_Adres_7_bit_2 : BOOL ;
   B_Adres_7_bit_3 : BOOL ;
   B_Adres_6_bit_0 : BOOL ;	//Temporary placeholder variable
   B_Adres_6_bit_1 : BOOL ;
   B_Adres_6_bit_2 : BOOL ;
   B_Adres_6_bit_3 : BOOL ;
   B_Adres_9_bit_0 : BOOL ;	//Temporary placeholder variable
   B_Adres_9_bit_1 : BOOL ;
   B_Adres_9_bit_2 : BOOL ;
   B_Adres_9_bit_3 : BOOL ;
   B_Adres_8_bit_0 : BOOL ;	//Temporary placeholder variable
   B_Adres_8_bit_1 : BOOL ;
   B_Adres_8_bit_2 : BOOL ;
   B_Adres_8_bit_3 : BOOL ;
   B_Adres_11_bit_0 : BOOL ;	//Temporary placeholder variable
   B_Adres_11_bit_1 : BOOL ;
   B_Adres_11_bit_2 : BOOL ;
   B_Adres_11_bit_3 : BOOL ;
   B_Adres_10_bit_0 : BOOL ;	//Temporary placeholder variable
   B_Adres_10_bit_1 : BOOL ;
   B_Adres_10_bit_2 : BOOL ;
   B_Adres_10_bit_3 : BOOL ;
   B_Adres_13_bit_0 : BOOL ;	//Temporary placeholder variable
   B_Adres_13_bit_1 : BOOL ;
   B_Adres_13_bit_2 : BOOL ;
   B_Adres_13_bit_3 : BOOL ;
   B_Adres_12_bit_0 : BOOL ;	//Temporary placeholder variable
   B_Adres_12_bit_1 : BOOL ;
   B_Adres_12_bit_2 : BOOL ;
   B_Adres_12_bit_3 : BOOL ;
   B_Adres_15_bit_0 : BOOL ;	//Temporary placeholder variable
   B_Adres_15_bit_1 : BOOL ;
   B_Adres_15_bit_2 : BOOL ;
   B_Adres_15_bit_3 : BOOL ;
   B_Adres_14_bit_0 : BOOL ;	//Temporary placeholder variable
   B_Adres_14_bit_1 : BOOL ;
   B_Adres_14_bit_2 : BOOL ;
   B_Adres_14_bit_3 : BOOL ;
   B_Adres_17_bit_0 : BOOL ;	//Temporary placeholder variable
   B_Adres_17_bit_1 : BOOL ;
   B_Adres_17_bit_2 : BOOL ;
   B_Adres_17_bit_3 : BOOL ;
   B_Adres_16_bit_0 : BOOL ;	//Temporary placeholder variable
   B_Adres_16_bit_1 : BOOL ;
   B_Adres_16_bit_2 : BOOL ;
   B_Adres_16_bit_3 : BOOL ;
   B_Adres_19_bit_0 : BOOL ;	//Temporary placeholder variable
   B_Adres_19_bit_1 : BOOL ;
   B_Adres_19_bit_2 : BOOL ;
   B_Adres_19_bit_3 : BOOL ;
   B_Adres_18_bit_0 : BOOL ;	//Temporary placeholder variable
   B_Adres_18_bit_1 : BOOL ;
   B_Adres_18_bit_2 : BOOL ;
   B_Adres_18_bit_3 : BOOL ;
   B_Adres_21_bit_0 : BOOL ;	//Temporary placeholder variable
   B_Adres_21_bit_1 : BOOL ;
   B_Adres_21_bit_2 : BOOL ;
   B_Adres_21_bit_3 : BOOL ;
   B_Adres_20_bit_0 : BOOL ;	//Temporary placeholder variable
   B_Adres_20_bit_1 : BOOL ;
   B_Adres_20_bit_2 : BOOL ;
   B_Adres_20_bit_3 : BOOL ;
   B_Adres_23_bit_0 : BOOL ;	//Temporary placeholder variable
   B_Adres_23_bit_1 : BOOL ;
   B_Adres_23_bit_2 : BOOL ;
   B_Adres_23_bit_3 : BOOL ;
   B_Adres_22_bit_0 : BOOL ;	//Temporary placeholder variable
   B_Adres_22_bit_1 : BOOL ;
   B_Adres_22_bit_2 : BOOL ;
   B_Adres_22_bit_3 : BOOL ;
   B_Adres_25_bit_0 : BOOL ;	//Temporary placeholder variable
   B_Adres_25_bit_1 : BOOL ;
   B_Adres_25_bit_2 : BOOL ;
   B_Adres_25_bit_3 : BOOL ;
   B_Adres_24_bit_0 : BOOL ;	//Temporary placeholder variable
   B_Adres_24_bit_1 : BOOL ;
   B_Adres_24_bit_2 : BOOL ;
   B_Adres_24_bit_3 : BOOL ;
   B_Adres_27_bit_0 : BOOL ;	//Temporary placeholder variable
   B_Adres_27_bit_1 : BOOL ;
   B_Adres_27_bit_2 : BOOL ;
   B_Adres_27_bit_3 : BOOL ;
   B_Adres_26_bit_0 : BOOL ;	//Temporary placeholder variable
   B_Adres_26_bit_1 : BOOL ;
   B_Adres_26_bit_2 : BOOL ;
   B_Adres_26_bit_3 : BOOL ;
   B_Adres_29_bit_0 : BOOL ;	//Temporary placeholder variable
   B_Adres_29_bit_1 : BOOL ;
   B_Adres_29_bit_2 : BOOL ;
   B_Adres_29_bit_3 : BOOL ;
   B_Adres_28_bit_0 : BOOL ;	//Temporary placeholder variable
   B_Adres_28_bit_1 : BOOL ;
   B_Adres_28_bit_2 : BOOL ;
   B_Adres_28_bit_3 : BOOL ;
   B_Adres_31_bit_0 : BOOL ;	//Temporary placeholder variable
   B_Adres_31_bit_1 : BOOL ;
   B_Adres_31_bit_2 : BOOL ;
   B_Adres_31_bit_3 : BOOL ;
   B_Adres_30_bit_0 : BOOL ;	//Temporary placeholder variable
   B_Adres_30_bit_1 : BOOL ;
   B_Adres_30_bit_2 : BOOL ;
   B_Adres_30_bit_3 : BOOL ;
  END_STRUCT ;	
BEGIN
END_DATA_BLOCK

DATA_BLOCK "MPI_GD"	// DB 100
VERSION : 0.1
  STRUCT
   IN : STRUCT
    Life_Bit_Foliarka : BOOL ;
    Foliarka_Automatyka : BOOL ;
    Foliarka_Reczny : BOOL ;
    Foto_Banda_1 : BOOL ;
    Foto_Owijarka : BOOL ;
    Rezerwa_1 : BOOL ;
    Motor_10_Lewo : BOOL ;	//przod
    Motor_10_Prawo : BOOL ;	//tyl
    Motor_11_Lewo : BOOL ;
    Motor_11_Prawo : BOOL ;
    Zezwolenie_Na_Wjazd_10 : BOOL ;
    Potw_Dost_Na_Wjazd_10 : BOOL ;
    Zabierz_Na_Bande_11 : BOOL ;
    Paleta_Obecna_Na_7_Tr : BOOL ;
    Paleta_Obraca_Sie : BOOL ;
    Foliowanie_Zakonczone : BOOL ;
    Banda_Fol_4_Foto_Tyl : BOOL ;
    Banda_Fol_4_Foto_Przod : BOOL ;
    Banda_Fol_4_Motor_Tyl : BOOL ;
    Banda_Fol_4_Motor_Przod : BOOL ;
    Banda_Fol_Obr_Foto_Tyl : BOOL ;	//Wirtualna fotokomorka tylna banda obr
    Banda_Fol_Obr_Foto_Przod : BOOL ;	//Wirtualna fotokomorka przod banda obr
    Banda_Fol_Obr_Motor_Tyl : BOOL ;
    Banda_Fol_Obr_Motor_Przo : BOOL ;
    Banda_Fol_6_Foto_Tyl : BOOL ;
    Banda_Fol_6_Foto_Przod : BOOL ;
    Banda_Fol_6_Motor_Tyl : BOOL ;
    Banda_Fol_6_Motor_Przod : BOOL ;
   END_STRUCT ;
   OUT : STRUCT
    Life_Bit_Szafa : BOOL ;
    Szafa_Automatyka : BOOL ;
    Foto_1_Banda_10 : BOOL ;	//przod
    Foto_2_Banda_10 : BOOL ;	//tyl
    Foto_Banda_11 : BOOL ;
    Silnik_10_OK : BOOL ;
    Silnik_11_OK : BOOL ;
    Zabierz_Na_Bande_10 : BOOL ;
    Zezwolenie_Na_Wyjazd_11 : BOOL ;
    Potw_Dost_Na_Wyjazd_11 : BOOL ;
    Obrot_Na_Poz_Wlot_1 : BOOL ;
    Zmien_Program_Na_4 : BOOL ;
    Zmien_Pragram_Na_3 : BOOL ;
    Foto_Banda_9 : BOOL ;
    Help_INT : INT ;
   END_STRUCT ;
  END_STRUCT ;	
BEGIN
END_DATA_BLOCK

